Aux_State_val := ck_state_v( Vision_struct.States_in);
//read register from robot and chek is can read 2 or more correct values 
IF Aux_State_val = VCts.SeparatorRot_L_I THEN
	 I_STATE:= VCts.SeparatorRot_L_I;
//verifies that the vision system has completed its task
ELSIF Aux_State_val = VCts.SeparatorRot_L_F THEN
	//read the values processed by the vision system and send to robot
	sep_rot_left_data := ck_real_value(Vision_struct.Head_left_value);
	//check if all values are correct
	//IF sep_rot_left_data.Flag THEN
		//write variables from PLC to CS.UR5 Robot
		//IF wr_real_value(VCts.HEAD_LEFT_VALUE,sep_rot_left_data.Value) THEN
		    wr_real_value(VCts.HEAD_LEFT_VALUE,sep_rot_left_data.Value);
			I_STATE := VCts.SeparatorRot_L_F;
		//END_IF
	//END_IF
	
END_IF


//read internal variable and write over output variable
Act_In_State := I_STATE;
END_ACTION

ACTION CkHeadRot_L_entry:
//start the vision system
wr_state_v(Vcts.SeparatorRot_L);

//write the retain state variable 
Act_Gl_State:=VCts.SeparatorRot_L;
END_ACTION

ACTION CkHeadRot_L_exit:
//write reset state variables to visiom system.
wr_state_v(RCts.RESET_STATE);
//reset Global state variable
G_STATE := -1;
I_STATE :=-1;

//reset flags vision system to PLC
Vision_struct.States_in.Val1 := -1;
Vision_struct.States_in.Val2 := -1;
Vision_struct.States_in.Val3 := -1;
END_ACTION

ACTION CkHole_active:

Aux_State_val := ck_state_v( Vision_struct.States_in);
//read register from robot and chek is can read 2 or more correct values 
IF Aux_State_val = VCts.SeparatorHole_I THEN
	 I_STATE:= VCts.SeparatorHole_I;
//verifies that the vision system has completed its task
ELSIF Aux_State_val = VCts.SeparatorHole_F THEN
	//read the values processed by the vision system and send to robot
	cx_vision_data := ck_real_value(Vision_struct.Cx_value_hole);
	cy_vision_data := ck_real_value(Vision_struct.Cy_value_hole);
	
	//check if all values are correct
//	IF cx_vision_data.Flag AND cy_vision_data.Flag THEN
//		//write variables from PLC to CS.UR5 Robot
//		IF wr_real_value(VCts.CX_VALUE,cx_vision_data.Value) THEN
//			IF wr_real_value(VCts.CY_VALUE,cy_vision_data.Value) THEN				
//						I_STATE := VCts.SeparatorHole_F;
//			END_IF
		
//		END_IF
//	END_IF
	wr_real_value(VCts.CX_VALUE,cx_vision_data.Value);
	wr_real_value(VCts.CY_VALUE,cy_vision_data.Value);
	I_STATE := VCts.SeparatorHole_F;
	
END_IF




//read internal variable and write over output variable
Act_In_State := I_STATE;
END_ACTION

ACTION CkHole_entry:
//start the vision system
wr_state_v(Vcts.SeparatorHole);

//write the retain state variable 
Act_Gl_State:=VCts.SeparatorHole;
END_ACTION

ACTION CkHole_exit:
//write reset state variables to visiom system.
wr_state_v(RCts.RESET_STATE);
//reset Global state variable
G_STATE := -1;
I_STATE :=-1;


//reset flags vision system to PLC
Vision_struct.States_in.Val1 := -1;
Vision_struct.States_in.Val2 := -1;
Vision_struct.States_in.Val3 := -1;
END_ACTION

ACTION CkNut_active:

Aux_State_val := ck_state_v( Vision_struct.States_in);
//read register from robot and chek is can read 2 or more correct values 
IF Aux_State_val = VCts.SeparatorNut_I THEN
	 I_STATE:= VCts.SeparatorNut_I;
//verifies that the vision system has completed its task
ELSIF Aux_State_val = VCts.SeparatorNut_F  THEN
	//read the values processed by the vision system and send to robot
	cx_vision_data := ck_real_value(Vision_struct.Cx_value_nut);
	cy_vision_data := ck_real_value(Vision_struct.Cy_value_nut);
	nut_turn_data := ck_real_value(Vision_struct.Nut_turn_value);
	//check if all values are correct
	//IF cx_vision_data.Flag AND cy_vision_data.Flag AND nut_turn_data.Flag THEN
		//write variables from PLC to CS.UR5 Robot
		//I_STATE := VCts.SeparatorNut_F;
		wr_real_value(VCts.CX_VALUE,cx_vision_data.Value);
		wr_real_value(VCts.CY_VALUE,cy_vision_data.Value);
		wr_real_value(VCts.NUT_VALUE,nut_turn_data.Value);
		I_STATE := VCts.SeparatorNut_F;
		
		//IF wr_real_value(VCts.CX_VALUE,cx_vision_data.Value) THEN
		//	IF wr_real_value(VCts.CY_VALUE,cy_vision_data.Value) THEN
			//	IF wr_real_value(VCts.NUT_VALUE,nut_turn_data.Value) THEN
			//			I_STATE := VCts.SeparatorNut_F;
			//	END_IF
			//END_IF
		
		//END_IF
		
	//END_IF
	
END_IF



//read internal variable and write over output variable
Act_In_State := I_STATE;
END_ACTION

ACTION CkNut_entry:
//start the vision system
wr_state_v(Vcts.SeparatorNut);

//write the retain state variable 
Act_Gl_State:=VCts.SeparatorNut;
END_ACTION

ACTION CkNut_exit:

//write reset state variables to visiom system.
wr_state_v(RCts.RESET_STATE);
//reset Global state variable
G_STATE := -1;
//rest internat state variable
I_STATE :=-1;

//reset flags vision system to PLC
Vision_struct.States_in.Val1 := -1;
Vision_struct.States_in.Val2 := -1;
Vision_struct.States_in.Val3 := -1;
END_ACTION

ACTION CkPosSep_active:

Aux_State_val := ck_state_v( Vision_struct.States_in);
//read register from robot and chek is can read 2 or more correct values 
IF Aux_State_val = VCts.SeparatorPos_I THEN
	 I_STATE:= VCts.SeparatorPos_I;
	
//verifies that the vision system has completed its task
ELSIF  Aux_State_val = VCts.SeparatorPos_F THEN
	//I_STATE := VCts.SeparatorPos_F;
	//read the values processed by the vision system and send to robot
	sep_pos_data := ck_real_value(Vision_struct.Pos_sep);
	//check if all values are correct
	//IF sep_pos_data.Flag THEN
		//write variables from PLC to CS.UR5 Robot
		//IF wr_real_value(VCts.SEP_POS_VALUE,sep_pos_data.Value) THEN
		wr_real_value(VCts.SEP_POS_VALUE,sep_pos_data.Value);
		I_STATE := VCts.SeparatorPos_F;

		//END_IF
	//END_IF
	
END_IF

//read internal variable and write over output variable
Act_In_State := I_STATE;
END_ACTION

ACTION CkPosSep_entry:

//start the vision system
wr_state_v(Vcts.SeparatorPos);

//write the retain state variable 
Act_Gl_State:=VCts.SeparatorPos;
END_ACTION

ACTION CkPosSep_exit:

//write reset state variables to visiom system.
wr_state_v(RCts.RESET_STATE);
//reset Global state variable
G_STATE := -1;
//rest internat state variable
I_STATE :=-1;

//reset flags vision system to PLC
Vision_struct.States_in.Val1 := -1;
Vision_struct.States_in.Val2 := -1;
Vision_struct.States_in.Val3 := -1;
END_ACTION

ACTION Wrt_FState_entry:
//write output variable to indicate that the robot execute the state 
State_complete := TRUE;
END_ACTION

ACTION Wrt_FState_exit:
//write output variable to indicate that the robot execute the state 
State_complete := FALSE;
//init_:=FALSE;

G_STATE := -1;
//rest internat state variable
I_STATE :=-1;
END_ACTION

END_PROGRAM

// ---- POUs/POUs/VISION/Vision_functions/ck_state_v.TcPOU
FUNCTION ck_state_v : INT
VAR_INPUT
	
	data_vision : Vision_int_state;
    
END_VAR
VAR
	ck0 : INT;
	ck1 : INT;
	ck2 : INT;
END_VAR


ck0 := data_vision.Val1;
ck1 := data_vision.Val2;
ck2 := data_vision.Val3;


//IF (ck0=state AND ck1=state AND ck2=state) OR (ck1=state AND ck2=state) OR (ck0=state AND ck2=state) OR (ck0=state AND ck1=state ) THEN
IF ck0 = ck1 THEN
ck_state_v := ck0;	
ELSIF  ck1 = ck2 THEN 
ck_state_v := ck1;	
ELSIF  ck2 = ck0 THEN
ck_state_v := ck2;	
ELSE 
ck_state_v := -1;	
END_IF

END_FUNCTION

// ---- POUs/POUs/VISION/Vision_functions/ck_real_value.TcPOU
FUNCTION ck_real_value :ck_real_flag_data
//return ck_real_flag_data struct
VAR_INPUT
	//imput Vision_data struct 
	data: Vision_data;
END_VAR
VAR
END_VAR


//check if two of tree values are the same, to avoid bad variables intercahnages between vision system and plc
//return flag ck_real_flag_data[0] to indicate is correct, and one real value ck_real_value[1] 
IF data.Val2=data.Val3 THEN
	ck_real_value.Flag:=TRUE;
	ck_real_value.Value:=data.Val2;
ELSIF data.Val1=data.Val3 THEN
	ck_real_value.Flag:=TRUE;
	ck_real_value.Value:=data.Val3;
ELSIF data.Val1=data.Val2 THEN
	ck_real_value.Flag:=TRUE;
	ck_real_value.Value:=data.Val2;
ELSIF (data.Val1=data.Val2 AND data.Val1=data.Val3 AND data.Val2=data.Val3) THEN	
	ck_real_value.Flag:=TRUE;
	ck_real_value.Value:=data.Val1;
ELSE	
	ck_real_value.Flag:=FALSE;
	ck_real_value.Value:=-1;
END_IF

END_FUNCTION

// ---- POUs/POUs/VISION/Vision_functions/wr_state_v.TcPOU
FUNCTION wr_state_v : BOOL
VAR_INPUT
	state : INT;
END_VAR
VAR
END_VAR

wr_state_v := FALSE;
//WRITE FLAGS STATE-MACHINE #################(PLC->VISION SYSTEM)
Vision_struct.States_out.Val1:=state;
Vision_struct.States_out.Val2:=state;
Vision_struct.States_out.Val3:=state;
wr_state_v := TRUE;

END_FUNCTION

// ---- POUs/POUs/Qrob/Qrob_State_Machine/QRob_StateMachine.TcPOU
PROGRAM QRob_StateMachine
VAR_INPUT
init_: BOOL:= True;
//global aux state
G_STATE : INT := -1;
//comaper position to stop
Position : LREAL:= 0;
Velocity : REAL:=170;
Torque : INT := 0;
Torque_ramp : INT := 100;
Control :E_DRIVEOPERATIONMODE;
Reset_State : BOOL:= FALSE;
//Max_profile_velocity AT%Q*:UDINT := 314572;
//Modes_operation AT%Q*:USINT:= 8;
//actual_torque AT%I*:INT ;

//Qrob_set torque 
torquevalut AT%Q*:INT;


END_VAR
VAR_OUTPUT
	State_complete : BOOL := FALSE;
	Act_Gl_State : INT := -1;
	Act_In_State : INT := -1;
	Act_Pos : LREAL := -1;
END_VAR
VAR
	
//Axis status
Axis_state :BOOL:=FALSE;
	//internal aux state
I_STATE : INT:=-1;
Aux_error :INT:=-1;
//blocks to activate axis of qrob
Reset : MC_Reset;
ResetOut: ST_McOutputs;

PowerAxis1 : MC_Power;
/// debug function block output data 
PowerAxis1Out: ST_McOutputs;



//blocks to move axis 
MoveAbsAxis1 :MC_MoveAbsolute;
MoveAbsoluteOut1: ST_McOutputs;

//block to set home position
Home : MC_Home;
HomeOut: ST_McOutputs;

//block to read and change the contyrol mode
WriteDriveOperationMode : MC_WriteDriveOperationMode;
WDO_ModeOut : ST_McOutputs;

ReadDriveOperationMode : MC_ReadDriveOperationMode;
RDO_ModeOut : ST_McOutputs;
ReadOperation_mode : E_DRIVEOPERATIONMODE;

//block to Control Mode
TorqueControl : MC_TorqueControl;
TorqueControlOut : ST_McOutputs;
Torque_done : BOOL;
Qrob_velocity AT%I*:DINT := -1;
Qrob_torque AT%I*:INT := -1;

//block stop motion
Stop : MC_Stop;
StopOut: ST_McOutputs;

//var to ck torque done
F_vel : BOOL ;
F_tor : BOOL;
F_tor_done : BOOL;


//var to offfset Home
offset_home :INT := 3;
offset_flag : INT := -1;

Sensor_Position_detection AT%I*: BOOL;


END_VAR

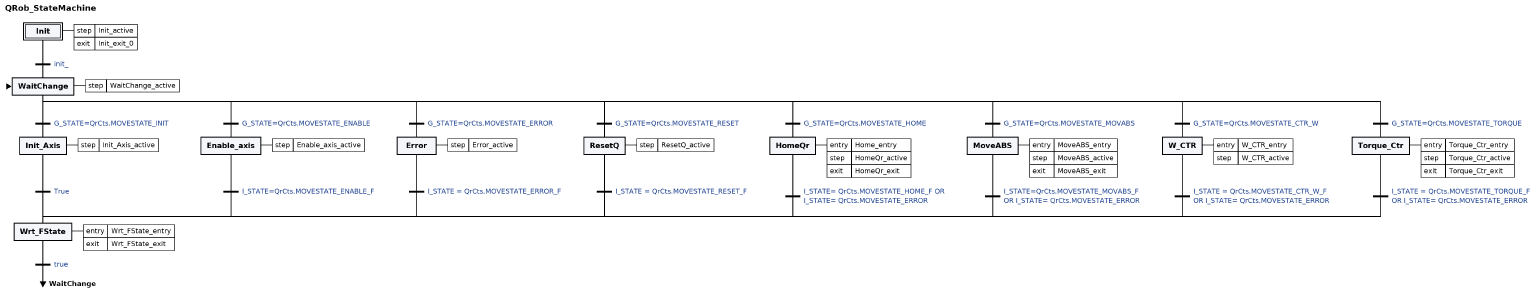
INITIAL_STEP Init:
    Init_active(N);  // step action
    Init_exit_0(P0);  // exit action
END_STEP
TRANSITION FROM Init TO WaitChange
    := init_;
END_TRANSITION
STEP WaitChange:
    WaitChange_active(N);  // step action
END_STEP
TRANSITION FROM WaitChange TO Init_Axis
    := G_STATE=QrCts.MOVESTATE_INIT;
END_TRANSITION
STEP Init_Axis:
    Init_Axis_active(N);  // step action
END_STEP
TRANSITION FROM Init_Axis TO Wrt_FState
    := True;
END_TRANSITION
TRANSITION FROM WaitChange TO Enable_axis
    := G_STATE=QrCts.MOVESTATE_ENABLE;
END_TRANSITION
STEP Enable_axis:
    Enable_axis_active(N);  // step action
END_STEP
TRANSITION FROM Enable_axis TO Wrt_FState
    := I_STATE=QrCts.MOVESTATE_ENABLE_F;
END_TRANSITION
TRANSITION FROM WaitChange TO Error
    := G_STATE=QrCts.MOVESTATE_ERROR;
END_TRANSITION
STEP Error:
    Error_active(N);  // step action
END_STEP
TRANSITION FROM Error TO Wrt_FState
    := I_STATE = QrCts.MOVESTATE_ERROR_F;
END_TRANSITION
TRANSITION FROM WaitChange TO ResetQ
    := G_STATE=QrCts.MOVESTATE_RESET;
END_TRANSITION
STEP ResetQ:
    ResetQ_active(N);  // step action
END_STEP
TRANSITION FROM ResetQ TO Wrt_FState
    := I_STATE = QrCts.MOVESTATE_RESET_F;
END_TRANSITION
TRANSITION FROM WaitChange TO HomeQr
    := G_STATE=QrCts.MOVESTATE_HOME;
END_TRANSITION
STEP HomeQr:
    Home_entry(P1);  // entry action
    HomeQr_active(N);  // step action
    HomeQr_exit(P0);  // exit action
END_STEP
TRANSITION FROM HomeQr TO Wrt_FState
    := I_STATE= QrCts.MOVESTATE_HOME_F OR I_STATE= QrCts.MOVESTATE_ERROR;
END_TRANSITION
TRANSITION FROM WaitChange TO MoveABS
    := G_STATE=QrCts.MOVESTATE_MOVABS;
END_TRANSITION
STEP MoveABS:
    MoveABS_entry(P1);  // entry action
    MoveABS_active(N);  // step action
    MoveABS_exit(P0);  // exit action
END_STEP
TRANSITION FROM MoveABS TO Wrt_FState
    := I_STATE=QrCts.MOVESTATE_MOVABS_F OR I_STATE= QrCts.MOVESTATE_ERROR;
END_TRANSITION
TRANSITION FROM WaitChange TO W_CTR
    := G_STATE=QrCts.MOVESTATE_CTR_W;
END_TRANSITION
STEP W_CTR:
    W_CTR_entry(P1);  // entry action
    W_CTR_active(N);  // step action
END_STEP
TRANSITION FROM W_CTR TO Wrt_FState
    := I_STATE = QrCts.MOVESTATE_CTR_W_F OR I_STATE= QrCts.MOVESTATE_ERROR;
END_TRANSITION
TRANSITION FROM WaitChange TO Torque_Ctr
    := G_STATE=QrCts.MOVESTATE_TORQUE;
END_TRANSITION
STEP Torque_Ctr:
    Torque_Ctr_entry(P1);  // entry action
    Torque_Ctr_active(N);  // step action
    Torque_Ctr_exit(P0);  // exit action
END_STEP
TRANSITION FROM Torque_Ctr TO Wrt_FState
    := I_STATE = QrCts.MOVESTATE_TORQUE_F OR I_STATE= QrCts.MOVESTATE_ERROR;
END_TRANSITION
STEP Wrt_FState:
    Wrt_FState_entry(P1);  // entry action
    Wrt_FState_exit(P0);  // exit action
END_STEP
TRANSITION FROM Wrt_FState TO WaitChange
    := true;
END_TRANSITION

ACTION AC_WriteControl:
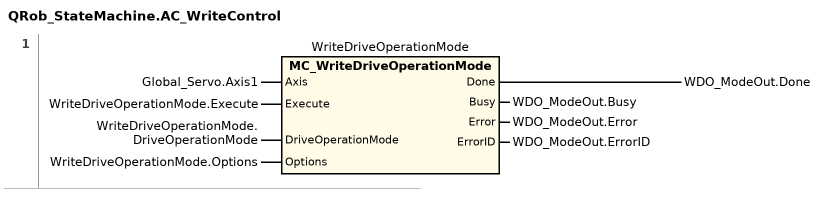
// NETWORK 1
WriteDriveOperationMode(
    Axis := Global_Servo.Axis1,
    Execute := WriteDriveOperationMode.Execute,
    DriveOperationMode := WriteDriveOperationMode.DriveOperationMode,
    Options := WriteDriveOperationMode.Options,
    Busy => WDO_ModeOut.Busy,
    Error => WDO_ModeOut.Error,
    ErrorID => WDO_ModeOut.ErrorID); // MC_WriteDriveOperationMode
WDO_ModeOut.Done := WriteDriveOperationMode.Done;
END_ACTION

ACTION Act_Home:
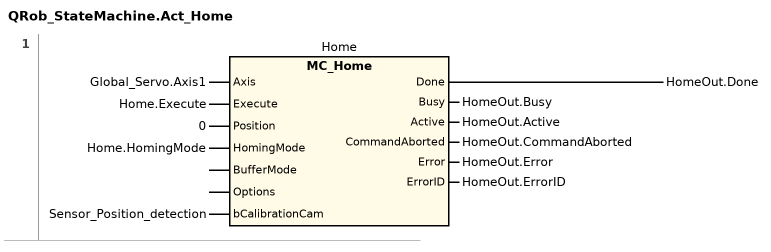
// NETWORK 1
Home(
    Axis := Global_Servo.Axis1,
    Execute := Home.Execute,
    Position := 0,
    HomingMode := Home.HomingMode,
    bCalibrationCam := Sensor_Position_detection,
    Busy => HomeOut.Busy,
    Active => HomeOut.Active,
    CommandAborted => HomeOut.CommandAborted,
    Error => HomeOut.Error,
    ErrorID => HomeOut.ErrorID); // MC_Home
HomeOut.Done := Home.Done;
END_ACTION

ACTION Act_MoveAbs:
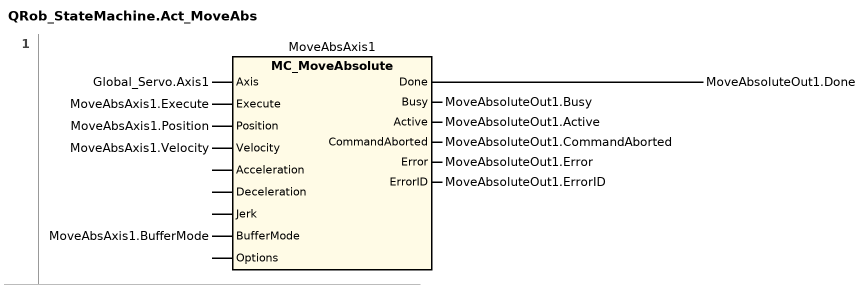
// NETWORK 1
MoveAbsAxis1(
    Axis := Global_Servo.Axis1,
    Execute := MoveAbsAxis1.Execute,
    Position := MoveAbsAxis1.Position,
    Velocity := MoveAbsAxis1.Velocity,
    BufferMode := MoveAbsAxis1.BufferMode,
    Busy => MoveAbsoluteOut1.Busy,
    Active => MoveAbsoluteOut1.Active,
    CommandAborted => MoveAbsoluteOut1.CommandAborted,
    Error => MoveAbsoluteOut1.Error,
    ErrorID => MoveAbsoluteOut1.ErrorID); // MC_MoveAbsolute
MoveAbsoluteOut1.Done := MoveAbsAxis1.Done;
END_ACTION

ACTION Act_Power:
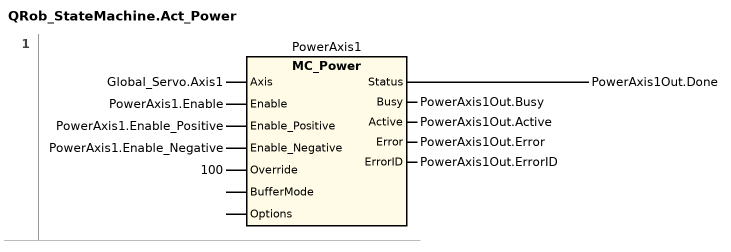
// NETWORK 1
PowerAxis1(
    Axis := Global_Servo.Axis1,
    Enable := PowerAxis1.Enable,
    Enable_Positive := PowerAxis1.Enable_Positive,
    Enable_Negative := PowerAxis1.Enable_Negative,
    Override := 100,
    Busy => PowerAxis1Out.Busy,
    Active => PowerAxis1Out.Active,
    Error => PowerAxis1Out.Error,
    ErrorID => PowerAxis1Out.ErrorID); // MC_Power
PowerAxis1Out.Done := PowerAxis1.Status;
END_ACTION

ACTION Act_ReadControl:
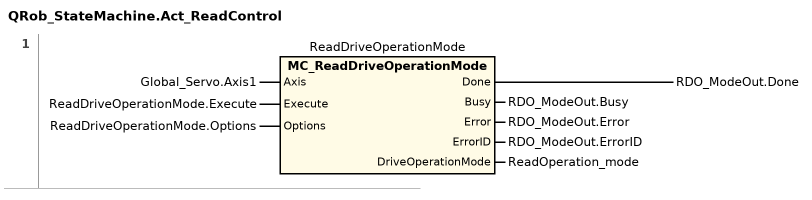
// NETWORK 1
ReadDriveOperationMode(
    Axis := Global_Servo.Axis1,
    Execute := ReadDriveOperationMode.Execute,
    Options := ReadDriveOperationMode.Options,
    Busy => RDO_ModeOut.Busy,
    Error => RDO_ModeOut.Error,
    ErrorID => RDO_ModeOut.ErrorID,
    DriveOperationMode => ReadOperation_mode); // MC_ReadDriveOperationMode
RDO_ModeOut.Done := ReadDriveOperationMode.Done;
END_ACTION

ACTION Act_Reset:
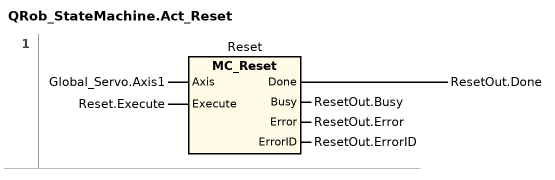
// NETWORK 1
Reset(
    Axis := Global_Servo.Axis1,
    Execute := Reset.Execute,
    Busy => ResetOut.Busy,
    Error => ResetOut.Error,
    ErrorID => ResetOut.ErrorID); // MC_Reset
ResetOut.Done := Reset.Done;
END_ACTION

ACTION Act_Stop:
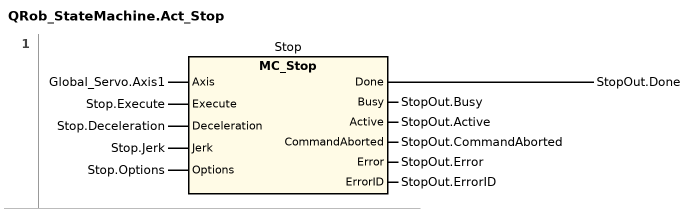
// NETWORK 1
Stop(
    Axis := Global_Servo.Axis1,
    Execute := Stop.Execute,
    Deceleration := Stop.Deceleration,
    Jerk := Stop.Jerk,
    Options := Stop.Options,
    Busy => StopOut.Busy,
    Active => StopOut.Active,
    CommandAborted => StopOut.CommandAborted,
    Error => StopOut.Error,
    ErrorID => StopOut.ErrorID); // MC_Stop
StopOut.Done := Stop.Done;
END_ACTION

ACTION Act_Torque:
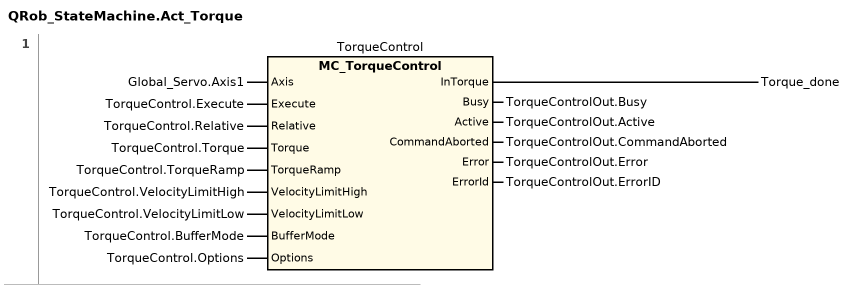
// NETWORK 1
TorqueControl(
    Axis := Global_Servo.Axis1,
    Execute := TorqueControl.Execute,
    Relative := TorqueControl.Relative,
    Torque := TorqueControl.Torque,
    TorqueRamp := TorqueControl.TorqueRamp,
    VelocityLimitHigh := TorqueControl.VelocityLimitHigh,
    VelocityLimitLow := TorqueControl.VelocityLimitLow,
    BufferMode := TorqueControl.BufferMode,
    Options := TorqueControl.Options,
    Busy => TorqueControlOut.Busy,
    Active => TorqueControlOut.Active,
    CommandAborted => TorqueControlOut.CommandAborted,
    Error => TorqueControlOut.Error,
    ErrorId => TorqueControlOut.ErrorID); // MC_TorqueControl
Torque_done := TorqueControl.InTorque;
END_ACTION

ACTION Enable_axis_active:
//power on axis
PowerAxis1.Enable := TRUE;
PowerAxis1.Enable_Positive := TRUE;
PowerAxis1.Enable_Negative := TRUE;


IF PowerAxis1.Status THEN
//check the state where the error is produced	
	CASE Aux_error OF 
		QrCts.MOVESTATE_MOVABS:
			G_STATE := QrCts.MOVESTATE_MOVABS;
		QrCts.MOVESTATE_HOME:
			G_STATE := QrCts.MOVESTATE_HOME;
		QrCts.MOVESTATE_CTR_W:
			G_STATE := QrCts.MOVESTATE_CTR_W;
		QrCts.MOVESTATE_TORQUE:	
			G_STATE := QrCts.MOVESTATE_TORQUE;
		QrCts.MOVESTATE_RELIEF:
			G_STATE := QrCts.MOVESTATE_RELIEF;
	ELSE
		G_STATE := -1;
	END_CASE
	I_STATE := QrCts.MOVESTATE_ENABLE_F;
ELSIF PowerAxis1.Error THEN
	G_STATE := QrCts.MOVESTATE_ERROR;
	I_STATE := QrCts.MOVESTATE_ENABLE_F;
END_IF

(* call the power function block *)
Act_Power();
Act_Reset();
Act_MoveAbs();
END_ACTION

ACTION Enable_axis_entry:
//power on axis
PowerAxis1.Enable := TRUE;
PowerAxis1.Enable_Positive := TRUE;
PowerAxis1.Enable_Negative := TRUE;
END_ACTION

ACTION Error_active:
IF Global_Servo.Axis1.NcToPlc.ErrorCode <>0 THEN
	G_STATE := QrCts.MOVESTATE_RESET;	(* axis error requires reset *)
	I_STATE := QrCts.MOVESTATE_ERROR_F;
ELSE
G_STATE := QrCts.MOVESTATE_INIT;
I_STATE := QrCts.MOVESTATE_ERROR_F;		(* function block errors don't need a reset *)
END_IF


(* call the power function block *)
Act_Power();
Act_Reset();
Act_MoveAbs();
END_ACTION

ACTION Home_entry:

//start fuction block 
Home.Execute := TRUE;

IF offset_flag = 1 THEN 
	Home.HomingMode := MC_Direct;
	offset_flag := offset_flag +1 ;
ELSE  	
	Home.HomingMode := MC_DefaultHoming;
END_IF


//write the retain state variable 
Act_Gl_State:=QrCts.MOVESTATE_HOME;
//read internal variable and write over output variable
I_STATE := QrCts.MOVESTATE_HOME_I;
Act_In_State := I_STATE;
END_ACTION

ACTION HomeQr_active:



//Home.bCalibrationCam := Sensor_Position_detection; 

IF Home.CommandAborted OR Home.Error THEN
	G_STATE := QrCts.MOVESTATE_ERROR;
	I_STATE := QrCts.MOVESTATE_ERROR;
	Aux_error := QrCts.MOVESTATE_HOME;
	Act_In_State := I_STATE;
ELSIF Home.Done THEN
	I_STATE := QrCts.MOVESTATE_HOME_F;
	//read internal variable and write over output variable
	Act_In_State := I_STATE;
	G_STATE := QrCts.MOVESTATE_MOVABS;
	position := offset_home;
	Home.Execute := FALSE; 
  IF offset_flag >= 2 THEN
	  G_STATE := -1;
	  offset_flag := -1;
  ELSE
	  G_STATE := QrCts.MOVESTATE_MOVABS;
	  offset_flag := offset_flag + 1;
  END_IF
	
END_IF





(* call the power function block *)
Act_Power();
Act_Reset();
Act_Home();
Act_MoveAbs();
END_ACTION

ACTION HomeQr_exit:
I_STATE :=-1;
END_ACTION

ACTION Init_active:

END_ACTION

ACTION Init_Axis_active:


//star variables
MoveAbsAxis1.Execute := FALSE;
Reset.Execute := FALSE;
Home.Execute := FALSE;
//write the global staus
G_State := QrCts.MOVESTATE_ENABLE;




(* call the power function block *)
Act_Power();
Act_Reset();
Act_MoveAbs();
Act_Home();
END_ACTION

ACTION Init_Axis_entry:

END_ACTION

ACTION Init_Axis_exit:

END_ACTION

ACTION Init_exit:
// NETWORK 1
END_ACTION

ACTION Init_exit_0:
G_STATE:=QrCts.MOVESTATE_INIT;


//check is there are some error
IF Global_Servo.Axis1.NcToPlc.ErrorCode <>0 THEN
	G_STATE := QrCts.MOVESTATE_RESET;	(* axis error requires reset *)
	
//ELSE
//	G_STATE := QrCts.MOVESTATE_INIT;
//	I_STATE := QrCts.MOVESTATE_ERROR_F;		(* function block errors don't need a reset *)
END_IF
END_ACTION

ACTION MoveABS_active:


IF MoveAbsAxis1.CommandAborted OR MoveAbsAxis1.Error THEN
	G_STATE := QrCts.MOVESTATE_ERROR;
	I_STATE := QrCts.MOVESTATE_ERROR;
	Aux_error := QrCts.MOVESTATE_MOVABS;
	Position := Position - Act_Pos;
	//read internal variable and write over output variable
	Act_In_State := I_STATE;
ELSIF MoveAbsAxis1.Done THEN
	I_STATE := QrCts.MOVESTATE_MOVABS_F;
	//read internal variable and write over output variable
	Act_In_State := I_STATE;
	G_STATE := -1;
	MoveAbsAxis1.Execute := FALSE;
ELSIF Reset_state THEN
	I_STATE := QrCts.MOVESTATE_MOVABS_F;;
	Act_In_State := I_STATE;
	G_STATE := -1;
	
	Stop.Execute := TRUE;
    MoveAbsAxis1.Execute := FALSE;	
	Reset_state := FALSE;
END_IF


//read actual postion
Act_Pos := Global_Servo.Axis1.NcToPlc.ActPos;

(* call the power function block *)
Act_Power();
Act_Reset();
Act_MoveAbs();
Act_Stop();
END_ACTION

ACTION MoveABS_entry:

MoveAbsAxis1.Position := Position;
MoveAbsAxis1.Velocity := Velocity;
//MoveAbsAxis1.BufferMode := MC_Buffered;
MoveAbsAxis1.Execute := TRUE;



//write the retain state variable 
Act_Gl_State:=QrCts.MOVESTATE_MOVABS;
//read internal variable and write over output variable
I_STATE := QrCts.MOVESTATE_MOVABS_I;
Act_In_State := I_STATE;

(* call the power function block *)
Act_Power();
Act_Reset();
Act_MoveAbs();
Act_Stop();
END_ACTION

ACTION MoveABS_exit:

//condition to execute home position
IF offset_flag = 0 THEN 
	G_STATE := QrCts.MOVESTATE_HOME;
    offset_flag := offset_flag +1 ;
END_IF


I_STATE :=-1;


Stop.Execute := FALSE;
Reset_state := FALSE;


(* call the power function block *)
Act_Power();
Act_Reset();
Act_MoveAbs();
Act_Stop();
END_ACTION

ACTION ResetQ_active:
WriteDriveOperationMode.Execute := FALSE;
Home.Execute := FALSE;
ReadDriveOperationMode.Execute := FALSE;
Stop.Execute := FALSE;
MoveAbsAxis1.Execute := FALSE;
TorqueControl.Execute := FALSE;
Stop.Execute := FALSE; 

Reset.Execute := TRUE;


IF Reset.Done THEN
	G_STATE := QrCts.MOVESTATE_INIT;
	I_STATE := QrCts.MOVESTATE_RESET_F;
ELSIF Reset.Error THEN
	G_STATE := QrCts.MOVESTATE_INIT; (* can't do anything here *)
	//I_STATE := QrCts.MOVESTATE_RESET_F;
END_IF


(* call the power function block *)
Act_Power();
Act_Reset();
Act_MoveAbs();
Act_Stop();
END_ACTION

ACTION Sleep_exit:
TorqueControl.Execute := False;
END_ACTION

ACTION Torque_Ctr_active:
IF TorqueControlOut.CommandAborted OR TorqueControlOut.Error THEN
	G_STATE := QrCts.MOVESTATE_ERROR;
	I_STATE := QrCts.MOVESTATE_ERROR;
	Aux_error := QrCts.MOVESTATE_TORQUE;
	//read internal variable and write over output variable
	Act_In_State := I_STATE;
ELSIF Torque_done THEN
	F_tor_done := TRUE;
END_IF



IF Qrob_torque = Torque THEN 
	F_tor := TRUE;
		IF Qrob_velocity <=0  THEN 
			F_vel := TRUE;
	END_IF
END_IF


IF F_vel AND F_tor AND F_tor_done THEN

	I_STATE := QrCts.MOVESTATE_TORQUE_F;
	//read internal variable and write over output variable
	Act_In_State := I_STATE;
	G_STATE := -1;
	TorqueControl.Execute := FALSE;
	Torque_done := FALSE;
	
	F_vel  := FALSE;
	F_tor  := FALSE;
	F_tor_done  := FALSE;
	//I_STATE :=-1;	

END_IF

(* call the power function block *)
Act_Power();
Act_Reset();
Act_MoveAbs();
Act_Torque();
END_ACTION

ACTION Torque_Ctr_entry:
// write the variables TorqueControl block function
TorqueControl.Relative := FALSE;
TorqueControl.Torque := Torque;
torquevalut := Torque;
TorqueControl.TorqueRamp := 100;
TorqueControl.VelocityLimitHigh := 100;
TorqueControl.VelocityLimitLow := 1;
TorqueControl.Execute := True;


//write the retain state variable 
Act_Gl_State:=QrCts.MOVESTATE_TORQUE;
//read internal variable and write over output variable
I_STATE := QrCts.MOVESTATE_TORQUE_I;
Act_In_State := I_STATE;
END_ACTION

ACTION Torque_Ctr_exit:
	TorqueControl.Execute := FALSE;
	Torque_done := FALSE;
	//I_STATE :=-1;
	//G_STATE := -1;
	
	I_STATE :=-1;
END_ACTION

ACTION Torque_Relie_active:
//ggggggggggggggg


IF TorqueControlOut.CommandAborted OR TorqueControlOut.Error THEN
	G_STATE := QrCts.MOVESTATE_ERROR;
	I_STATE := QrCts.MOVESTATE_ERROR;
	Aux_error := QrCts.MOVESTATE_RELIEF;
	//read internal variable and write over output variable
	Act_In_State := I_STATE;
ELSIF Torque_done THEN
	F_tor_done := TRUE;
END_IF

//F_tor_done := TRUE;

IF Qrob_torque = 0 THEN 
	F_tor := TRUE;
		IF (-5 <= Qrob_velocity) AND  (Qrob_velocity<= 5) THEN 
			F_vel := TRUE;
	END_IF
END_IF


IF F_vel AND F_tor AND F_tor_done THEN

	I_STATE := QrCts.MOVESTATE_RELIEF_F;
	//read internal variable and write over output variable
	Act_In_State := I_STATE;
	G_STATE := -1;
	TorqueControl.Execute := TRUE;
	Torque_done := FALSE;
	
	F_vel  := FALSE;
	F_tor  := FALSE;
	F_tor_done  := FALSE;
	//I_STATE :=-1;	

END_IF

(* call the power function block *)
Act_Power();
Act_Reset();
Act_MoveAbs();
Act_Torque();
END_ACTION

ACTION Torque_Relie_entry:
// write the variables TorqueControl block function
TorqueControl.Relative := FALSE;
TorqueControl.Torque := 0;
TorqueControl.TorqueRamp := 0;
TorqueControl.VelocityLimitHigh := 100;
TorqueControl.VelocityLimitLow := 0;
//torquevalut := 0;
TorqueControl.Execute := True;


//write the retain state variable 
Act_Gl_State:=QrCts.MOVESTATE_RELIEF;
//read internal variable and write over output variable
I_STATE := QrCts.MOVESTATE_RELIEF_I;
Act_In_State := I_STATE;
END_ACTION

ACTION Torque_Relie_exit:
	TorqueControl.Execute := FALSE;
	Torque_done := FALSE;
	
	I_STATE :=-1;
END_ACTION

ACTION W_CTR_active:
IF WriteDriveOperationMode.Error THEN
	G_STATE := QrCts.MOVESTATE_ERROR;
	I_STATE := QrCts.MOVESTATE_ERROR;
	Aux_error := QrCts.MOVESTATE_CTR_W;
	//read internal variable and write over output variable
	Act_In_State := I_STATE;
ELSIF WriteDriveOperationMode.Done THEN
	//Read if the control mode have been change
	ReadDriveOperationMode.Execute := TRUE;
	IF ReadDriveOperationMode.Error THEN
		G_STATE := QrCts.MOVESTATE_ERROR;
		I_STATE := QrCts.MOVESTATE_ERROR;
		Aux_error := QrCts.MOVESTATE_CTR_W;
		//read internal variable and write over output variable
		Act_In_State := I_STATE;
	 	ReadDriveOperationMode.Execute := FALSE; 
	
	ELSIF ReadDriveOperationMode.Done THEN
		
		IF ReadOperation_mode = Control THEN

			I_STATE := QrCts.MOVESTATE_CTR_W_F;
			//read internal variable and write over output variable
			Act_In_State := I_STATE;
			//G_STATE := -1;
			WriteDriveOperationMode.Execute := FALSE;
			ReadDriveOperationMode.Execute := FALSE; 
			G_STATE := QrCts.MOVESTATE_RESET;
			//I_STATE :=-1;
		END_IF
		ReadDriveOperationMode.Execute := FALSE; 
	END_IF
END_IF


(* call the  function block *)
Act_Power();
Act_Reset();
AC_WriteControl();
Act_ReadControl();
END_ACTION

ACTION W_CTR_entry:
WriteDriveOperationMode.DriveOperationMode := Control;
WriteDriveOperationMode.Execute := TRUE;

//write the retain state variable 
Act_Gl_State:=QrCts.MOVESTATE_CTR_W;
//read internal variable and write over output variable
I_STATE := QrCts.MOVESTATE_CTR_W_I;
Act_In_State := I_STATE;
END_ACTION

ACTION WaitChange_active:

END_ACTION

ACTION Wrt_FState_entry:
//write output variable to indicate that the robot execute the state 
State_complete := TRUE;
END_ACTION

ACTION Wrt_FState_exit:
//write output variable to indicate that the robot execute the state 
State_complete := FALSE;
Reset_State := FALSE;
END_ACTION

END_PROGRAM

// ---- POUs/POUs/ROBOTS/Robot_functions/read_bool_flag_move.TcPOU
FUNCTION read_bool_flag_move : BOOL
VAR_INPUT

	state : BOOL;
END_VAR
VAR
	ck0 : BOOL;
	ck1 : BOOL;
	ck2 : BOOL;
END_VAR

//Read bit register from Robot to PLC
ck0 := Robot_UR5.UR_outputs.B3;
ck1 := Robot_UR5.UR_outputs.B4;
ck2 := Robot_UR5.UR_outputs.B5;

IF (ck0=state AND ck1=state AND ck2=state) OR (ck0<>state AND ck1=state AND ck2=state) OR (ck0=state AND ck1<>state AND ck2=state) OR (ck0=state AND ck1=state AND ck2<>state) THEN
read_bool_flag_move := TRUE;
ELSE 
read_bool_flag_move := FALSE;	
END_IF

END_FUNCTION

// ---- POUs/POUs/ROBOTS/Robot_functions/read_bool_flag.TcPOU
FUNCTION read_bool_flag : BOOL
VAR_INPUT

	state : BOOL;
END_VAR
VAR
	ck0 : BOOL;
	ck1 : BOOL;
	ck2 : BOOL;
END_VAR

//Read bit register from Robot to PLC
ck0 := Robot_UR5.UR_outputs.B0;
ck1 := Robot_UR5.UR_outputs.B1;
ck2 := Robot_UR5.UR_outputs.B2;

IF (ck0=state AND ck1=state AND ck2=state) OR (ck0<>state AND ck1=state AND ck2=state) OR (ck0=state AND ck1<>state AND ck2=state) OR (ck0=state AND ck1=state AND ck2<>state) THEN
read_bool_flag := TRUE;
ELSE 
read_bool_flag := FALSE;	
END_IF

END_FUNCTION

// ---- POUs/POUs/Qrob/QRob_functions/Get_QRob_Pos.TcPOU
PROGRAM Get_QRob_Pos
VAR
	
MC_ReadActualPosition : MC_ReadActualPosition;
actual_position : REAL;

Driver_temperature_C AT%I*:UINT:= 0;


    FB_CoERead_ByDriveRef : FB_CoERead_ByDriveRef;
    stDriveRef        :  ST_DriveRef := (sNetId:= '172.18.236.0.6.1', nDriveNo := 1, nDriveType := 16, nSlaveAddr := 1001); 

    Index             : WORD := 16#22A2;
    SubIndex          : BYTE := 0; 
    Execute           : BOOL := TRUE;
    Timeout           : TIME := T#5S;
    CompleteAccess    : BOOL := TRUE;
    vendorId          : UINT ;
    Error             : BOOL;
    AdsErrId          : UDINT;
    CANopenErrId      : UDINT;
	
	FB_EcCoESdoRead : FB_EcCoESdoRead;
	dir :  T_AmsNetId := '172.18.236.0.6.1';
	
	pSample : POINTER TO UINT;
	driver_temperature : UINT;
	
	Cooler_fan AT%Q*:BOOL:= FALSE;
	Temperature_Ctr : Temperature_Ctr;

END_VAR

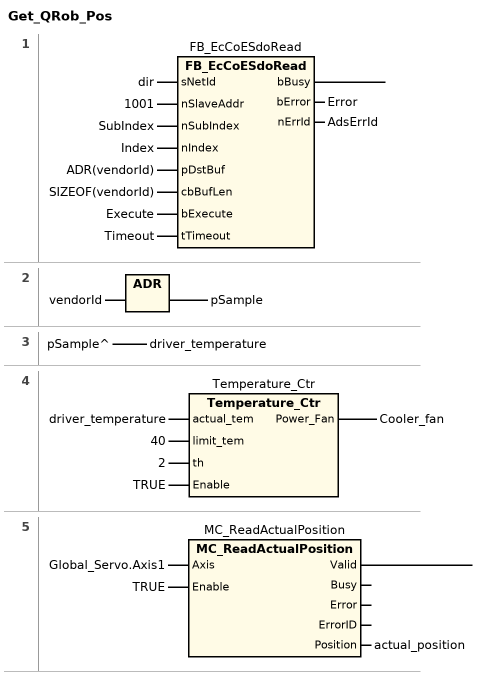
// NETWORK 1
FB_EcCoESdoRead(
    sNetId := dir,
    nSlaveAddr := 1001,
    nSubIndex := SubIndex,
    nIndex := Index,
    pDstBuf := ADR(vendorId),
    cbBufLen := SIZEOF(vendorId),
    bExecute := Execute,
    tTimeout := Timeout,
    bError => Error,
    nErrId => AdsErrId);

// NETWORK 2
pSample := ADR(vendorId);

// NETWORK 3
driver_temperature := pSample^;

// NETWORK 4
Temperature_Ctr(actual_tem := driver_temperature, limit_tem := 40, th := 2, Enable := TRUE);
Cooler_fan := Temperature_Ctr.Power_Fan;

// NETWORK 5
MC_ReadActualPosition(Axis := Global_Servo.Axis1, Enable := TRUE, Position => actual_position);

END_PROGRAM

// ---- POUs/POUs/Qrob/QRob_functions/Temperature_Ctr.TcPOU
FUNCTION_BLOCK Temperature_Ctr
VAR_INPUT
	actual_tem : REAL;
	limit_tem : REAL;
	th : REAL;
	Enable : BOOL;	
	
	//relief_turn : BOOL := FALSE;	
   
	
END_VAR
VAR_OUTPUT
	Power_Fan :BOOL;
END_VAR
VAR
	A : REAL;
	B : REAL;
	
END_VAR


IF Enable = TRUE THEN 
	A := limit_tem-th;
	B := limit_tem +th;
	
	IF (actual_tem <= A)  THEN 
		Power_Fan := FALSE;
	ELSIF (actual_tem >= B) THEN
		Power_Fan := TRUE;
	END_IF
END_IF

END_FUNCTION_BLOCK

// ---- POUs/POUs/Fuzzy/Subsystem.TcPOU
FUNCTION_BLOCK Subsystem
VAR_INPUT
	in: LREAL;
	state : BOOL;
END_VAR
VAR_OUTPUT
	out: LREAL;
	set_move  : BOOL := TRUE;
	
END_VAR
VAR
	
  	state_aux : BOOL := FALSE;	
	before_out : INT;
	aux : INT := 0;
out_int : INT;


	ruleID: DINT;
	y1: LREAL;
	y2: LREAL;
	outputMFCache: ARRAY[0..302] OF LREAL;
	sampleID: DINT;
	rtb_antecedentOutputs: ARRAY[0..2] OF LREAL;
	rtb_aggregatedOutputs: ARRAY[0..100] OF LREAL;
	tmp: ARRAY[0..100] OF LREAL;
	tmp_0: ARRAY[0..100] OF LREAL;
	tmp_1: ARRAY[0..100] OF LREAL;
	inputMFCache_idx_1: LREAL;
	inputMFCache_idx_2: LREAL;
	i0_trimf_l: trimf_l;
	OutputSamplePoints_Value: ARRAY[0..100] OF LREAL := [0.0, 1.5, 3.0, 4.5, 6.0, 7.5, 9.0, 10.5, 12.0, 13.5, 15.0, 16.5, 18.0, 19.5, 21.0, 22.5, 24.0, 25.5, 27.0, 28.5, 30.0, 31.5, 33.0, 34.5, 36.0, 37.5, 39.0, 40.5, 42.0, 43.5, 45.0, 46.5, 48.0, 49.5, 51.0, 52.5, 54.0, 55.5, 57.0, 58.5, 60.0, 61.5, 63.0, 64.5, 66.0, 67.5, 69.0, 70.5, 72.0, 73.5, 75.0, 76.5, 78.0, 79.5, 81.0, 82.5, 84.0, 85.5, 87.0, 88.5, 90.0, 91.5, 93.0, 94.5, 96.0, 97.5, 99.0, 100.5, 102.0, 103.5, 105.0, 106.5, 108.0, 109.5, 111.0, 112.5, 114.0, 115.5, 117.0, 118.5, 120.0, 121.5, 123.0, 124.5, 126.0, 127.5, 129.0, 130.5, 132.0, 133.5, 135.0, 136.5, 138.0, 139.5, 141.0, 142.5, 144.0, 145.5, 147.0, 148.5, 150.0];
	c: ARRAY[0..2] OF LREAL := [21.73, 73.97, 122.6];
	b: ARRAY[0..2] OF LREAL := [54.58, 118.2, 170.8];
	b_c: ARRAY[0..2] OF LREAL := [-66.3, -24.7, 15.5325443786982];
	b_d: ARRAY[0..2] OF LREAL := [4.2869822485207, 56.4869822485207, 90.1869822485207];
	e: ARRAY[0..2] OF LREAL := [73.88, 114.1, 158.0];
	b_b: ARRAY[0..2] OF SINT := [3, 3, 1];
	
	
	

END_VAR


VAR RETAIN
    nRem1 : INT :=0;
END_VAR


(* Outputs for Atomic SubSystem: '<Root>/Subsystem' *)
(* Outputs for Atomic SubSystem: '<S1>/FuzzzyCtr' *)
(* MATLAB Function: '<S2>/Evaluate Rule Antecedents' *)
(* MATLAB Function 'Evaluate Rule Antecedents': '<S4>:1' *)
(* '<S4>:1:4' if SimulateUsing==1 &amp;&amp; coder.internal.canUseExtrinsic ... *)
(* '<S4>:1:5'         &amp;&amp; (isa(inputs,'double') || isa(inputs,'single')) *)
(* '<S4>:1:32' else *)
(* '<S4>:1:33' if fis.inputFuzzySetType==1 *)
(* '<S4>:1:34' [antecedentOutputs,sumAntecedentOutputs] = ... *)
(* '<S4>:1:35'             fuzzy.internal.codegen.evaluateRuleAntecedent(... *)
(* '<S4>:1:36'             inputs,fis,diagnostics); *)
y1 := 0.0;
y2 := 0.0;

IF in >= -17.61 THEN 
    y1 := 1.0;
END_IF;


IF in < -77.61 THEN 
    y1 := 0.0;
END_IF;


IF (-77.61 <= in) AND (in < -17.61) THEN 
    y1 := (in - -77.61) * 0.016666666666666666;
END_IF;


IF in <= 4.584 THEN 
    y2 := 1.0;
END_IF;


IF in > 31.8 THEN 
    y2 := 0.0;
END_IF;


IF (4.584 < in) AND (in <= 31.8) THEN 
    y2 := (31.8 - in) * 0.036743092298647854;
END_IF;

y1 := MIN(y1, y2);
inputMFCache_idx_1 := trimf(x := in, params1 := c);
inputMFCache_idx_2 := trimf(x := in, params1 := b);

IF 1.0 <= y1 THEN 
    y1 := 1.0;
END_IF;

y2 := y1;
rtb_antecedentOutputs[0] := y1;

IF 1.0 > inputMFCache_idx_1 THEN 
    y1 := inputMFCache_idx_1;
ELSE 
    y1 := 1.0;
END_IF;

y2 := y2 + y1;
rtb_antecedentOutputs[1] := y1;

IF 1.0 > inputMFCache_idx_2 THEN 
    y1 := inputMFCache_idx_2;
ELSE 
    y1 := 1.0;
END_IF;

y2 := y2 + y1;
rtb_antecedentOutputs[2] := y1;
(* MATLAB Function: '<S2>/Evaluate Rule Consequents' incorporates:
 *  Constant: '<S2>/Output Sample Points' *)
(* MATLAB Function 'Evaluate Rule Consequents': '<S5>:1' *)
(* '<S5>:1:4' if SimulateUsing==1 &amp;&amp; coder.internal.canUseExtrinsic ... *)
(* '<S5>:1:5'         &amp;&amp; (isa(inputs,'double') || isa(inputs,'single')) *)
(* '<S5>:1:55' else *)
(* '<S5>:1:56' if fis.inputFuzzySetType==1 *)
(* '<S5>:1:57' if strcmp(char(fis.type),'mamdani') *)
(* '<S5>:1:58' aggregatedOutputs = ... *)
(* '<S5>:1:59'                 fuzzy.internal.codegen.evaluateRuleConsequentForMamdaniFIS(... *)
(* '<S5>:1:60'                 antecedentOutputs,fis,samplePoints); *)
i0_trimf_l(x := OutputSamplePoints_Value, params1 := b_c);
tmp := i0_trimf_l.y;
i0_trimf_l(x := OutputSamplePoints_Value, params1 := b_d);
tmp_0 := i0_trimf_l.y;
i0_trimf_l(x := OutputSamplePoints_Value, params1 := e);
tmp_1 := i0_trimf_l.y;
(* End of Outputs for SubSystem: '<S1>/FuzzzyCtr' *)
(* End of Outputs for SubSystem: '<Root>/Subsystem' *)
(* Outputs for Atomic SubSystem: '<Root>/Subsystem' *)
(* Outputs for Atomic SubSystem: '<S1>/FuzzzyCtr' *)
(* MATLAB Function: '<S2>/Evaluate Rule Consequents' *)

FOR ruleID := 0 TO 100 DO 
    rtb_aggregatedOutputs[ruleID] := 0.0;
    outputMFCache[3 * ruleID] := tmp[ruleID];
    outputMFCache[(3 * ruleID) + 1] := tmp_0[ruleID];
    outputMFCache[(3 * ruleID) + 2] := tmp_1[ruleID];
END_FOR;


FOR ruleID := 0 TO 2 DO 
    inputMFCache_idx_1 := rtb_antecedentOutputs[ruleID];

    FOR sampleID := 0 TO 100 DO 
        inputMFCache_idx_2 := rtb_aggregatedOutputs[sampleID];
        y1 := outputMFCache[((3 * sampleID) + SINT_TO_DINT(b_b[ruleID])) - 1];

        IF y1 > inputMFCache_idx_1 THEN 
            y1 := inputMFCache_idx_1;
        END_IF;


        IF inputMFCache_idx_2 < y1 THEN 
            inputMFCache_idx_2 := y1;
        END_IF;

        rtb_aggregatedOutputs[sampleID] := inputMFCache_idx_2;
    END_FOR;

END_FOR;

(* MATLAB Function: '<S2>/Defuzzify Outputs' incorporates:
 *  Constant: '<S2>/Output Sample Points'
 *  MATLAB Function: '<S2>/Evaluate Rule Antecedents' *)
(* MATLAB Function 'Defuzzify Outputs': '<S3>:1' *)
(* '<S3>:1:4' if SimulateUsing==1 &amp;&amp; coder.internal.canUseExtrinsic ... *)
(* '<S3>:1:5'         &amp;&amp; (isa(aggregatedOutputs,'double') || isa(aggregatedOutputs,'single')) *)
(* '<S3>:1:63' else *)
(* '<S3>:1:64' if fis.inputFuzzySetType==1 *)
(* '<S3>:1:65' if isequal(fis.type,uint8('mamdani')) *)
(* '<S3>:1:66' defuzzifiedOutputs = ... *)
(* '<S3>:1:67'                 fuzzy.internal.codegen.applyMamdaniDefuzzificationMethod(... *)
(* '<S3>:1:68'                 samplePoints,sumAntecedentOutputs,aggregatedOutputs, ... *)
(* '<S3>:1:69'                 fis,diagnostics); *)

IF y2 = 0.0 THEN 
    (* Outport: '<Root>/out' *)
    out := 75.0;
ELSE 
    y2 := 0.0;
    y1 := 0.0;

    FOR ruleID := 0 TO 100 DO 
        y1 := y1 + rtb_aggregatedOutputs[ruleID];
    END_FOR;


    IF y1 = 0.0 THEN 
        (* Outport: '<Root>/out' *)
        out := 75.0;
    ELSE 

        FOR ruleID := 0 TO 100 DO 
            y2 := (OutputSamplePoints_Value[ruleID] * rtb_aggregatedOutputs[ruleID]) + y2;
        END_FOR;

        (* Outport: '<Root>/out' incorporates:
         *  Constant: '<S2>/Output Sample Points' *)
        out := (1.0 / y1) * y2;
    END_IF;

END_IF;

out_int := LREAL_TO_INT(out);

IF in>= Qrob_control.limite_corriente THEN 
 out := 0;	
 state_aux := TRUE;
END_IF

IF state_aux THEN
	//out := 0;
	//state_aux := FALSE;
END_IF

set_move := TRUE;
IF state THEN 
	set_move := FALSE;
END_IF
	
	



nRem1 := out_int;
(* End of MATLAB Function: '<S2>/Defuzzify Outputs' *)
(* End of Outputs for SubSystem: '<S1>/FuzzzyCtr' *)
(* End of Outputs for SubSystem: '<Root>/Subsystem' *)

END_FUNCTION_BLOCK

// ---- POUs/POUs/Fuzzy/trimf_l.TcPOU
FUNCTION_BLOCK trimf_l
VAR_INPUT
	x: ARRAY[0..100] OF LREAL;
	params1: ARRAY[0..2] OF LREAL;
END_VAR
VAR_OUTPUT
	y: ARRAY[0..100] OF LREAL;
END_VAR
VAR
	a: LREAL;
	b: LREAL;
	c: LREAL;
	i: DINT;
	x_0: LREAL;
END_VAR


a := params1[0];
b := params1[1];
c := params1[2];

FOR i := 0 TO 100 DO 
    x_0 := x[i];
    y[i] := 0.0;

    IF a <> b THEN 

        IF a < x_0 THEN 

            IF x_0 < b THEN 
                y[i] := (1.0 / (b - a)) * (x_0 - a);
            END_IF;

        END_IF;

    END_IF;


    IF b <> c THEN 

        IF b < x_0 THEN 

            IF x_0 < c THEN 
                y[i] := (1.0 / (c - b)) * (c - x_0);
            END_IF;

        END_IF;

    END_IF;


    IF x_0 = b THEN 
        y[i] := 1.0;
    END_IF;

END_FOR;

END_FUNCTION_BLOCK

// ---- POUs/POUs/Fuzzy/trimf.TcPOU
FUNCTION trimf : LREAL
VAR_INPUT
	x: LREAL;
	params1: ARRAY[0..2] OF LREAL;
END_VAR
VAR
END_VAR


trimf := 0.0;

IF params1[0] <> params1[1] THEN 

    IF params1[0] < x THEN 

        IF x < params1[1] THEN 
            trimf := (1.0 / (params1[1] - params1[0])) * (x - params1[0]);
        END_IF;

    END_IF;

END_IF;


IF params1[1] <> params1[2] THEN 

    IF params1[1] < x THEN 

        IF x < params1[2] THEN 
            trimf := (1.0 / (params1[2] - params1[1])) * (params1[2] - x);
        END_IF;

    END_IF;

END_IF;


IF x = params1[1] THEN 
    trimf := 1.0;
END_IF;

END_FUNCTION

// ---- POUs/POUs/Qrob/QRob_functions/Qrob_control.TcPOU
PROGRAM Qrob_control

VAR_INPUT
	


	torque_set_point AT%Q*:INT;
	torque_enable : BOOL := FALSE;
	enable_torque_out :BOOL;
	torque_decre : REAL :=2;
	
	torque_max_vel : REAL := 200;
	
	actual_torque AT%I*:INT ;
	actual_velocity : REAL;
	done_torqte_lib : BOOL;
	t_aux : INT;
	start_plot : BOOL;
	aux_cu :REAL;
	bthome : BOOL;
	home :	 BOOL;
	reset : bool;
	external : BOOL;
    mover_horario:	BOOL;
	mover_antihorario: BOOL;
	velocidad: REAL := 10 ;
	velocidad_ext: REAL := 100 ;
	set_posicion_mover :INT := 25;
	EnableAxis1 : BOOL := TRUE;
	detener : BOOL;
	mover_abs :BOOL;
	pos_mover_abs :REAL ;
	

	
	
	ajustar_tornillo : BOOL ;
	limite_corriente : REAL := 120;
	torque_relief : BOOL := FALSE;
	tor_on : BOOL;
    tor_val : INT;
		aux_velo : BOOL;
	
END_VAR

VAR
	MC_BufferMode :MC_BufferMode;
	fbPower: MC_Power;
	Axis1Enabled : BOOL;
	actual_position : LREAL;
	//actual_velocity : REAL;
	original_vel :DINT;
	actual_current  :  LREAL;
	position_ok :BOOL;
	
	mov_abs_ok : BOOL;
	max_current : BOOL;
	val_max_current : REAL;
	aux_current : REAL;

	
	MC_Home: MC_HOME;
	MC_ReadActualPosition: MC_ReadActualPosition;
	MC_ReadActualVelocity : MC_ReadActualVelocity;
	MC_ReadParameter_0: MC_ReadParameter;
	MC_MoveVelocity_horario: MC_MoveVelocity;
	MC_MoveVelocity_antiorario: MC_MoveVelocity;
	MC_Stop: MC_Stop;
	MC_Stop2: MC_Stop;
	MC_MoveAbsolute: MC_MoveAbsolute;
    MC_TorqueControl : MC_TorqueControl;
	Ton : TON;
	RS : RS;
	limit_current : limit_current;
	
	
	fuzzy : Subsystem;
	fuzzy_vel : LREAL;
	fuzzy_active : BOOL;
	stop_limit : BOOL;
    MC_ExtSetPointGenEnable : MC_ExtSetPointGenEnable;
	MC_Reset : MC_Reset;
	MC_MoveSuperImposed : MC_MoveSuperImposed;
    FB_CTRL_SETPOINT_GENERATOR : FB_CTRL_SETPOINT_GENERATOR;

	num_ran : LREAL;
	pulse : BOOL:= TRUE;
	PT_b : BOOL;
	DRAND : DRAND;
	pulse1 : pulse_;
	nrand_out : LREAL;
   
	state_move_active : BOOL;	


Max_profile_velocity AT%Q*:UDINT := 314572;
Modes_operation AT%Q*:USINT:= 8;

END_VAR

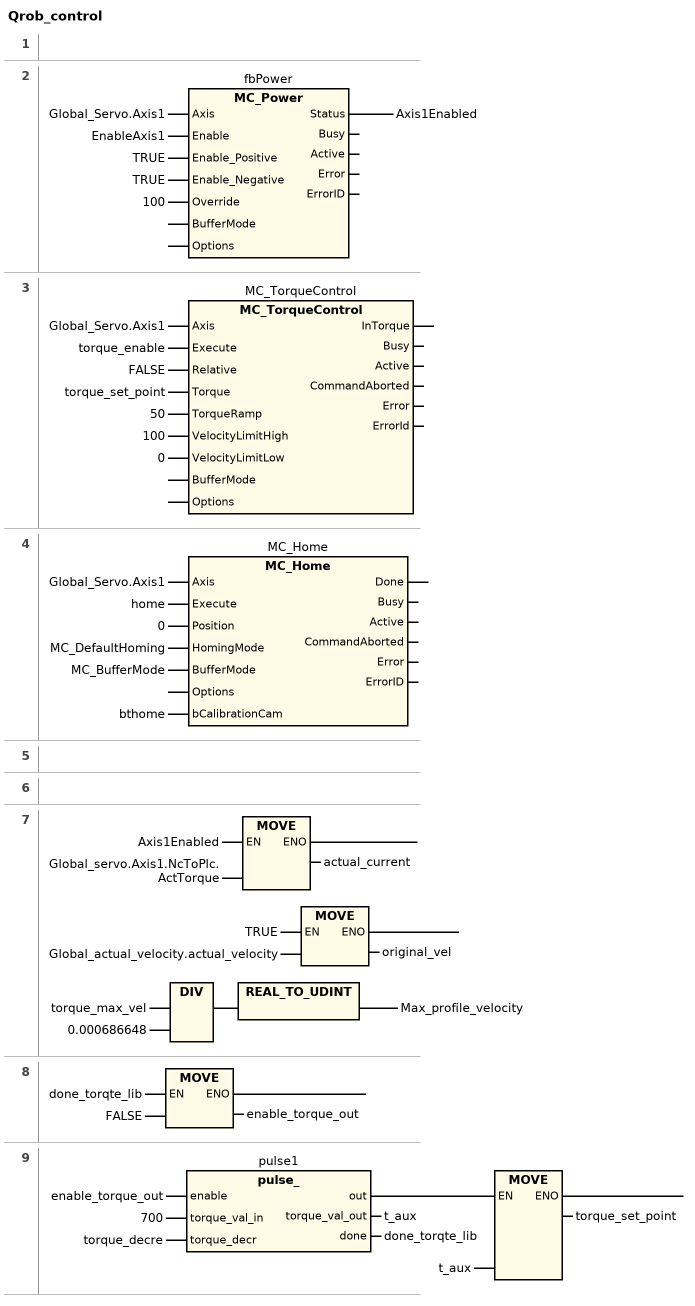
// NETWORK 1

// NETWORK 2
fbPower(
    Axis := Global_Servo.Axis1,
    Enable := EnableAxis1,
    Enable_Positive := TRUE,
    Enable_Negative := TRUE,
    Override := 100); // MC_Power
Axis1Enabled := fbPower.Status;

// NETWORK 3
MC_TorqueControl(
    Axis := Global_Servo.Axis1,
    Execute := torque_enable,
    Relative := FALSE,
    Torque := torque_set_point,
    TorqueRamp := 50,
    VelocityLimitHigh := 100,
    VelocityLimitLow := 0);

// NETWORK 4
MC_Home(
    Axis := Global_Servo.Axis1,
    Execute := home,
    Position := 0,
    HomingMode := MC_DefaultHoming,
    BufferMode := MC_BufferMode,
    bCalibrationCam := bthome);

// NETWORK 5

// NETWORK 6

// NETWORK 7
IF Axis1Enabled THEN actual_current := Global_servo.Axis1.NcToPlc.ActTorque; END_IF
original_vel := Global_actual_velocity.actual_velocity;
Max_profile_velocity := REAL_TO_UDINT(torque_max_vel / 0.000686648);

// NETWORK 8
IF done_torqte_lib THEN enable_torque_out := FALSE; END_IF

// NETWORK 9
pulse1(
    enable := enable_torque_out,
    torque_val_in := 700,
    torque_decr := torque_decre,
    torque_val_out => t_aux,
    done => done_torqte_lib); // pulse_
IF pulse1.out THEN torque_set_point := t_aux; END_IF

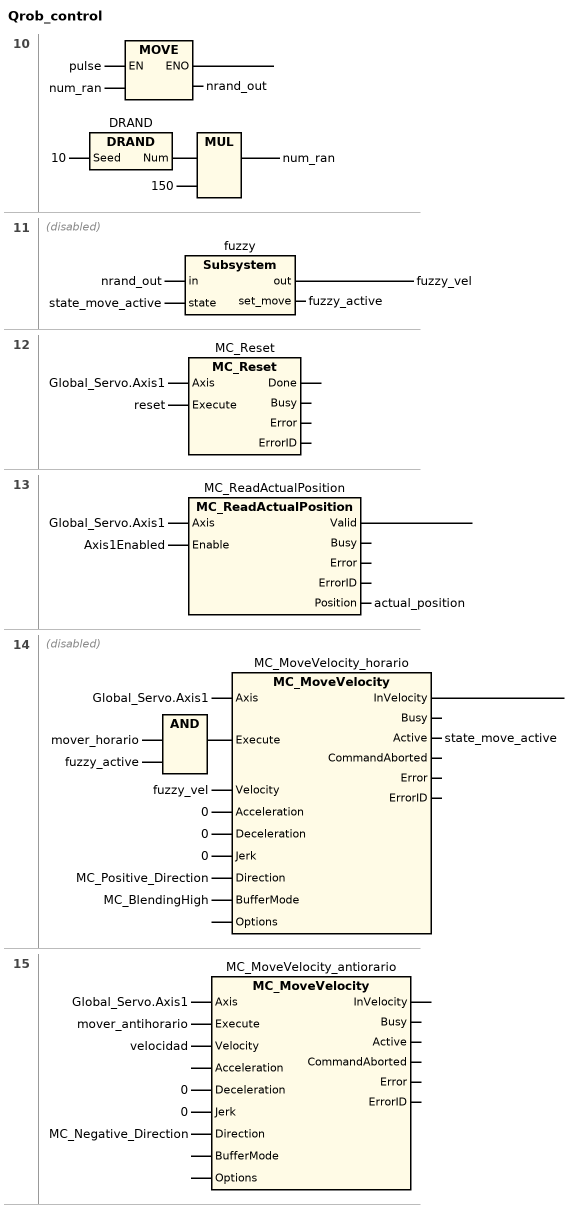
// NETWORK 10
IF pulse THEN nrand_out := num_ran; END_IF
DRAND(Seed := 10);
num_ran := DRAND.Num * 150;

// NETWORK 11 (disabled)
// fuzzy(in := nrand_out, state := state_move_active, set_move => fuzzy_active); // Subsystem
// fuzzy_vel := fuzzy.out;

// NETWORK 12
MC_Reset(Axis := Global_Servo.Axis1, Execute := reset);

// NETWORK 13
MC_ReadActualPosition(Axis := Global_Servo.Axis1, Enable := Axis1Enabled, Position => actual_position);

// NETWORK 14 (disabled)
// MC_MoveVelocity_horario(
//     Axis := Global_Servo.Axis1,
//     Execute := mover_horario AND fuzzy_active,
//     Velocity := fuzzy_vel,
//     Acceleration := 0,
//     Deceleration := 0,
//     Jerk := 0,
//     Direction := MC_Positive_Direction,
//     BufferMode := MC_BlendingHigh,
//     Active => state_move_active); // MC_MoveVelocity

// NETWORK 15
MC_MoveVelocity_antiorario(
    Axis := Global_Servo.Axis1,
    Execute := mover_antihorario,
    Velocity := velocidad,
    Deceleration := 0,
    Jerk := 0,
    Direction := MC_Negative_Direction); // MC_MoveVelocity

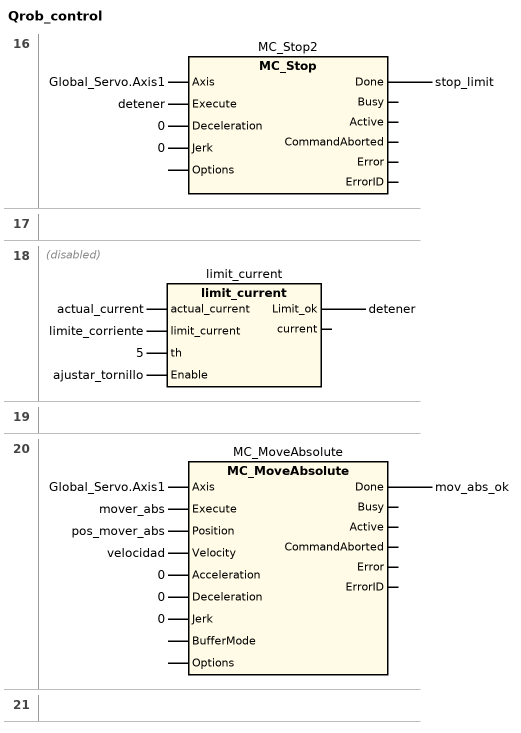
// NETWORK 16
MC_Stop2(Axis := Global_Servo.Axis1, Execute := detener, Deceleration := 0, Jerk := 0); // MC_Stop
stop_limit := MC_Stop2.Done;

// NETWORK 17

// NETWORK 18 (disabled)
// limit_current(
//     actual_current := actual_current,
//     limit_current := limite_corriente,
//     th := 5,
//     Enable := ajustar_tornillo);
// detener := limit_current.Limit_ok;

// NETWORK 19

// NETWORK 20
MC_MoveAbsolute(
    Axis := Global_Servo.Axis1,
    Execute := mover_abs,
    Position := pos_mover_abs,
    Velocity := velocidad,
    Acceleration := 0,
    Deceleration := 0,
    Jerk := 0);
mov_abs_ok := MC_MoveAbsolute.Done;

// NETWORK 21

END_PROGRAM

// ---- POUs/POUs/l/limit_current.TcPOU
FUNCTION_BLOCK limit_current
VAR_INPUT
	actual_current : REAL;
	limit_current : REAL;
	th : REAL;
	Enable : BOOL;	
	
	//relief_turn : BOOL := FALSE;	
   
	
END_VAR
VAR_OUTPUT
	Limit_ok :BOOL;
	current : REAL;
END_VAR
VAR
	A : REAL;
	B : REAL;
	
END_VAR


IF Enable = TRUE THEN 
	A := limit_current-th;
	B := limit_current +th;
	
	IF (A <= actual_current) AND (actual_current <= B) THEN 
		current := actual_current;
		IF current >= limit_current THEN
		  Limit_ok := TRUE;			 
		END_IF

	END_IF
ELSE
	 Limit_ok := FALSE;
	
END_IF

END_FUNCTION_BLOCK

// ---- POUs/POUs/l/pulse_.TcPOU
FUNCTION_BLOCK pulse_
VAR_INPUT
	enable: BOOL:= FALSE;
	torque_val_in : INT;
	torque_decr : REAL:= 2;
END_VAR
VAR_OUTPUT
	out: BOOL:= FALSE;
	torque_val_out :INT;
	done :BOOL;
	
END_VAR
VAR
	torque_aux : REAL;
END_VAR

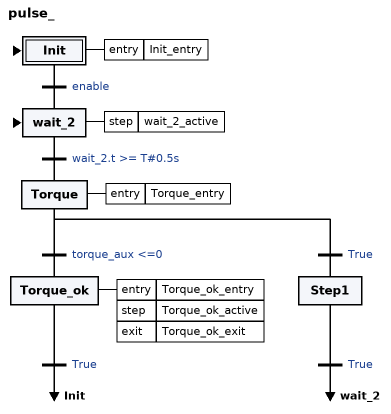
INITIAL_STEP Init:
    Init_entry(P1);  // entry action
END_STEP
TRANSITION FROM Init TO wait_2
    := enable;
END_TRANSITION
STEP wait_2:
    wait_2_active(N);  // step action
END_STEP
TRANSITION FROM wait_2 TO Torque
    := wait_2.t >= T#0.5s;
END_TRANSITION
STEP Torque:
    Torque_entry(P1);  // entry action
END_STEP
TRANSITION FROM Torque TO Torque_ok
    := torque_aux <=0;
END_TRANSITION
STEP Torque_ok:
    Torque_ok_entry(P1);  // entry action
    Torque_ok_active(N);  // step action
    Torque_ok_exit(P0);  // exit action
END_STEP
TRANSITION FROM Torque_ok TO Init
    := True;
END_TRANSITION
TRANSITION FROM Torque TO Step1
    := True;
END_TRANSITION
STEP Step1:
END_STEP
TRANSITION FROM Step1 TO wait_2
    := True;
END_TRANSITION

ACTION Init_entry:
out := FALSE;
done := False;
torque_aux := torque_val_in;
END_ACTION

ACTION Torque_entry:
torque_aux:=  ((torque_aux/torque_decr));


IF torque_aux <0 THEN
	torque_aux :=0 ;
END_IF

IF enable = TRUE THEN
torque_val_out := REAL_TO_INT(torque_aux);
END_IF
END_ACTION

ACTION Torque_ok_active:

END_ACTION

ACTION Torque_ok_entry:
out := TRUE;
done := TRue;
END_ACTION

ACTION Torque_ok_exit:
out:=FALSE;
END_ACTION

ACTION wait_1_active:
out := False;
END_ACTION

ACTION wait_2_active:
out := True;
END_ACTION

END_FUNCTION_BLOCK

// ---- POUs/POUs/IR_take_img/get_images.TcPOU
PROGRAM get_images
VAR
	start_head: BOOL;
	start_nut : BOOL;
	vi_get_img_cabezal_dere : BOOL;
	vi_get_img_nut : BOOL;
	head_ok : BOOL;
	nut_ok : BOOL;
END_VAR

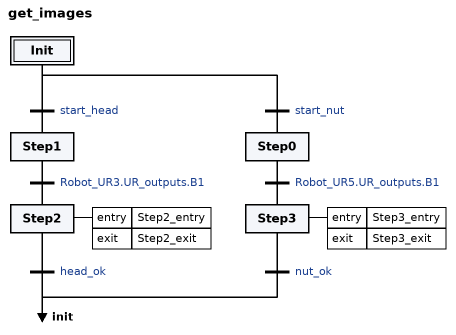
INITIAL_STEP Init:
END_STEP
TRANSITION FROM Init TO Step1
    := start_head;
END_TRANSITION
STEP Step1:
END_STEP
TRANSITION FROM Step1 TO Step2
    := Robot_UR3.UR_outputs.B1;
END_TRANSITION
STEP Step2:
    Step2_entry(P1);  // entry action
    Step2_exit(P0);  // exit action
END_STEP
TRANSITION FROM Step2 TO init
    := head_ok;
END_TRANSITION
TRANSITION FROM Init TO Step0
    := start_nut;
END_TRANSITION
STEP Step0:
END_STEP
TRANSITION FROM Step0 TO Step3
    := Robot_UR5.UR_outputs.B1;
END_TRANSITION
STEP Step3:
    Step3_entry(P1);  // entry action
    Step3_exit(P0);  // exit action
END_STEP
TRANSITION FROM Step3 TO init
    := nut_ok;
END_TRANSITION

ACTION Step2_entry:
vi_get_img_cabezal_dere := TRUE;
Robot_UR3.UR_inputs.Bits.B1 := False;
END_ACTION

ACTION Step2_exit:
vi_get_img_cabezal_dere := FALSE;
Robot_UR3.UR_inputs.Bits.B1 := TRUE;
head_ok := False;
END_ACTION

ACTION Step3_entry:
vi_get_img_nut := TRUE;
Robot_UR5.UR_inputs.Bits.B1 := False;
END_ACTION

ACTION Step3_exit:
vi_get_img_nut := FALSE;
Robot_UR5.UR_inputs.Bits.B1 := TRUE;
nut_ok := False;
END_ACTION

END_PROGRAM

// ---- POUs/POUs/l/Atornillar_ur5.TcPOU
PROGRAM Atornillar_UR5
VAR
END_VAR

VAR_INPUT
	Iniciar : Bool;
	Corriente : REAL :=10;
	Vueltas : REAL := 1;
	giro_alivio : LREAL := 0;
END_VAR
VAR_OUTPUT
END_VAR
VAR
	cal_vueltas : REAL;
	ct : INT;
	TIME_IN :TIME := T#10000MS;
	wait_t : BOOL;
END_VAR

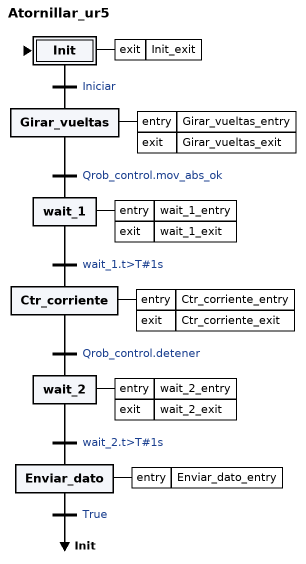
INITIAL_STEP Init:
    Init_exit(P0);  // exit action
END_STEP
TRANSITION FROM Init TO Girar_vueltas
    := Iniciar;
END_TRANSITION
STEP Girar_vueltas:
    Girar_vueltas_entry(P1);  // entry action
    Girar_vueltas_exit(P0);  // exit action
END_STEP
TRANSITION FROM Girar_vueltas TO wait_1
    := Qrob_control.mov_abs_ok;
END_TRANSITION
STEP wait_1:
    wait_1_entry(P1);  // entry action
    wait_1_exit(P0);  // exit action
END_STEP
TRANSITION FROM wait_1 TO Ctr_corriente
    := wait_1.t>T#1s;
END_TRANSITION
STEP Ctr_corriente:
    Ctr_corriente_entry(P1);  // entry action
    Ctr_corriente_exit(P0);  // exit action
END_STEP
TRANSITION FROM Ctr_corriente TO wait_2
    := Qrob_control.detener;
END_TRANSITION
STEP wait_2:
    wait_2_entry(P1);  // entry action
    wait_2_exit(P0);  // exit action
END_STEP
TRANSITION FROM wait_2 TO Enviar_dato
    := wait_2.t>T#1s;
END_TRANSITION
STEP Enviar_dato:
    Enviar_dato_entry(P1);  // entry action
END_STEP
TRANSITION FROM Enviar_dato TO Init
    := True;
END_TRANSITION

ACTION Alivio_torque_entry:
//regreo un grado para aliviar el torque y que pueda salir la herramienta
//Robot_A.UR_inputs.Bits.B11 := TRUE;
//wait_t := FALSE;
//Qrob_control.pos_mover_abs := Qrob_control.actual_position - giro_alivio;
//Qrob_control.velocidad := 50;
//Qrob_control.mover_abs := TRUE;


//Qrob_control.ajustar_tornillo := TRUE;
//Qrob_control.torque_relief := TRUE;
//Qrob_control.pos_mover_abs := Qrob_control.actual_position - giro_alivio;
//Qrob_control.velocidad := 0.5;
//Qrob_control.limite_corriente := 10;
//Qrob_control.mover_abs := TRUE;
END_ACTION

ACTION Alivio_torque_exit:

Robot_UR5.UR_inputs.Bits.B10 := FALSE;
//Qrob_control.ajustar_tornillo := FALSE;
//Qrob_control.torque_relief := FALSE;
Qrob_control.mover_abs := FALSE;
Qrob_control.detener := TRUE;
Qrob_control.detener := FALSE;
END_ACTION

ACTION Ctr_corriente_entry:
//cuando haya llegado al numero de vueltas especificado , realizo control de corriente 

wait_t := FALSE;
//FOR ct:=1 TO 5000 BY 1 DO
//Qrob_control.velocidad := 20;  
//END_FOR;

Qrob_control.ajustar_tornillo := TRUE;
Qrob_control.pos_mover_abs := 5000000;	
Qrob_control.velocidad := 100;
Qrob_control.limite_corriente := Corriente;
Qrob_control.mover_abs := TRUE;
END_ACTION

ACTION Ctr_corriente_exit:

Qrob_control.ajustar_tornillo := FALSE;
Qrob_control.detener := TRUE;
Qrob_control.detener := FALSE;
Qrob_control.mover_abs := FALSE;
END_ACTION

ACTION Enviar_dato_entry:

Robot_UR5.UR_inputs.Bits.B7 := TRUE;
Global_servo.Atornillado_ok :=TRUE;
END_ACTION

ACTION Girar_vueltas_entry:
// muevo ciertas cantidas d evuelatas a mayor velocidad y sin control de corriente 
Qrob_control.ajustar_tornillo := FALSE;


cal_vueltas := Qrob_control.actual_position + vueltas*360;
Qrob_control.pos_mover_abs := cal_vueltas;	
Qrob_control.velocidad := 180;
Qrob_control.mover_abs := TRUE;
END_ACTION

ACTION Girar_vueltas_exit:
Qrob_control.detener := TRUE;
Qrob_control.detener := FALSE;
Qrob_control.mover_abs := FALSE;
END_ACTION

ACTION Init_exit:

Robot_UR5.UR_inputs.Bits.B7 := FALSE;
Robot_UR5.UR_inputs.Bits.B8 := FALSE;
Iniciar := False;
END_ACTION

ACTION wait_1_entry:
Robot_UR5.UR_inputs.Bits.B10 := TRUE;
Qrob_control.detener := TRUE;
Qrob_control.detener := FALSE;
Qrob_control.mover_abs := FALSE;
END_ACTION

ACTION wait_1_exit:
Robot_UR5.UR_inputs.Bits.B10 := FALSE;
END_ACTION

ACTION wait_2_entry:


Qrob_control.detener := TRUE;
Qrob_control.detener := FALSE;
Qrob_control.mover_abs := FALSE;

Robot_UR5.UR_inputs.Bits.B7 := True;
END_ACTION

ACTION wait_2_exit:
Robot_UR5.UR_inputs.Bits.B7 := FALSE;
END_ACTION

END_PROGRAM

// ---- POUs/POUs/l/data_robot_ur5.TcPOU
PROGRAM data_robot_UR5
VAR
	
join_pos_1 : REAL;
join_pos_2 : REAL;
join_pos_3 : REAL;
join_pos_4 : REAL;
join_pos_5 : REAL;
join_pos_6 : REAL;

join_torque_1: REAL;
join_torque_2: REAL;
join_torque_3: REAL;
join_torque_4: REAL;
join_torque_5: REAL;
join_torque_6: REAL;

TCP_pos_x : REAL;
TCP_pos_y : REAL;
TCP_pos_z : REAL;
TCP_pos_rx : REAL;
TCP_pos_ry : REAL;
TCP_pos_rz : REAL;


TCP_force_x : REAL;
TCP_force_y : REAL;
TCP_force_z : REAL;
TCP_torque_x : REAL;
TCP_torque_y : REAL;
TCP_torque_z : REAL;

TCP_force : REAL;
velocity :INT;
turn_aux_float : REAL:= 0;
turn_aux_int : INT := 0;
qRob_actual_pos : REAL;	
new_turn : REAL;

//velocity_degress : REAL;
END_VAR


qRob_actual_pos := Get_QRob_Pos.actual_position/360;
turn_aux_int := ABS(REAL_TO_INT(qRob_actual_pos));
turn_aux_float:= turn_aux_int  - (qRob_actual_pos);
new_turn := turn_aux_float*(-1)*360;

TCP_pos_x := flip_byte(Robot_UR5.UR_TCP.FLOAT0)*1000;
TCP_pos_y := flip_byte(Robot_UR5.UR_TCP.FLOAT1)*1000;
TCP_pos_z := flip_byte(Robot_UR5.UR_TCP.FLOAT2)*1000;
TCP_pos_rx := (flip_byte(Robot_UR5.UR_TCP.FLOAT3)*180)/3.1415;
TCP_pos_ry := (flip_byte(Robot_UR5.UR_TCP.FLOAT4)*180)/3.1415;
TCP_pos_rz := (flip_byte(Robot_UR5.UR_TCP.FLOAT5)*180)/3.1415;


TCP_force  := flip_byte(Robot_UR5.UR_TCP.FLOAT18);

TCP_force_x := flip_byte(Robot_UR5.UR_TCP.FLOAT12);
TCP_force_y := flip_byte(Robot_UR5.UR_TCP.FLOAT13);
TCP_force_z := flip_byte(Robot_UR5.UR_TCP.FLOAT14);
TCP_torque_x := flip_byte(Robot_UR5.UR_TCP.FLOAT15);
TCP_torque_y := flip_byte(Robot_UR5.UR_TCP.FLOAT16);
TCP_torque_z := flip_byte(Robot_UR5.UR_TCP.FLOAT17);

join_pos_1 := (flip_byte(Robot_UR5.UR_JOINS.FLOAT0)*180)/3.1415;
join_pos_2 := (flip_byte(Robot_UR5.UR_JOINS.FLOAT1)*180)/3.1415;
join_pos_3 := (flip_byte(Robot_UR5.UR_JOINS.FLOAT2)*180)/3.1415;
join_pos_4 := (flip_byte(Robot_UR5.UR_JOINS.FLOAT3)*180)/3.1415;
join_pos_5 := (flip_byte(Robot_UR5.UR_JOINS.FLOAT4)*180)/3.1415;
join_pos_6 := (flip_byte(Robot_UR5.UR_JOINS.FLOAT5)*180)/3.1415;
 
join_torque_1 := flip_byte(Robot_UR5.UR_float_out.FLOAT0);
join_torque_2 := flip_byte(Robot_UR5.UR_float_out.FLOAT1);
join_torque_3 := flip_byte(Robot_UR5.UR_float_out.FLOAT2);
join_torque_4 := flip_byte(Robot_UR5.UR_float_out.FLOAT3);
join_torque_5 := flip_byte(Robot_UR5.UR_float_out.FLOAT4);
join_torque_6 := flip_byte(Robot_UR5.UR_float_out.FLOAT5);

END_PROGRAM

// ---- POUs/POUs/l/data_robot_ur3.TcPOU
PROGRAM data_robot_ur3





VAR
	
join_pos_1 : REAL;
join_pos_2 : REAL;
join_pos_3 : REAL;
join_pos_4 : REAL;
join_pos_5 : REAL;
join_pos_6 : REAL;

join_torque_1: REAL;
join_torque_2: REAL;
join_torque_3: REAL;
join_torque_4: REAL;
join_torque_5: REAL;
join_torque_6: REAL;

TCP_pos_x : REAL;
TCP_pos_y : REAL;
TCP_pos_z : REAL;
TCP_pos_rx : REAL;
TCP_pos_ry : REAL;
TCP_pos_rz : REAL;


TCP_force_x : REAL;
TCP_force_y : REAL;
TCP_force_z : REAL;
TCP_torque_x : REAL;
TCP_torque_y : REAL;
TCP_torque_z : REAL;

TCP_force : REAL;

END_VAR





TCP_pos_x := flip_byte(Robot_UR3.UR_TCP.FLOAT0)*1000;
TCP_pos_y := flip_byte(Robot_UR3.UR_TCP.FLOAT1)*1000;
TCP_pos_z := flip_byte(Robot_UR3.UR_TCP.FLOAT2)*1000;
TCP_pos_rx := (flip_byte(Robot_UR3.UR_TCP.FLOAT3)*180)/PI;
TCP_pos_ry := (flip_byte(Robot_UR3.UR_TCP.FLOAT4)*180)/PI;
TCP_pos_rz := (flip_byte(Robot_UR3.UR_TCP.FLOAT5)*180)/PI;


TCP_force  := flip_byte(Robot_UR3.UR_TCP.FLOAT18);

TCP_force_x := flip_byte(Robot_UR3.UR_TCP.FLOAT12);
TCP_force_y := flip_byte(Robot_UR3.UR_TCP.FLOAT13);
TCP_force_z := flip_byte(Robot_UR3.UR_TCP.FLOAT14);
TCP_torque_x := flip_byte(Robot_UR3.UR_TCP.FLOAT15);
TCP_torque_y := flip_byte(Robot_UR3.UR_TCP.FLOAT16);
TCP_torque_z := flip_byte(Robot_UR3.UR_TCP.FLOAT17);

join_pos_1 := (flip_byte(Robot_UR3.UR_JOINS.FLOAT0)*180)/PI;
join_pos_2 := (flip_byte(Robot_UR3.UR_JOINS.FLOAT1)*180)/PI;
join_pos_3 := (flip_byte(Robot_UR3.UR_JOINS.FLOAT2)*180)/PI;
join_pos_4 := (flip_byte(Robot_UR3.UR_JOINS.FLOAT3)*180)/PI;
join_pos_5 := (flip_byte(Robot_UR3.UR_JOINS.FLOAT4)*180)/PI;
join_pos_6 := (flip_byte(Robot_UR3.UR_JOINS.FLOAT5)*180)/PI;
 
join_torque_1 := flip_byte(Robot_UR3.UR_float_out.FLOAT0);
join_torque_2 := flip_byte(Robot_UR3.UR_float_out.FLOAT1);
join_torque_3 := flip_byte(Robot_UR3.UR_float_out.FLOAT2);
join_torque_4 := flip_byte(Robot_UR3.UR_float_out.FLOAT3);
join_torque_5 := flip_byte(Robot_UR3.UR_float_out.FLOAT4);
join_torque_6 := flip_byte(Robot_UR3.UR_float_out.FLOAT5);

END_PROGRAM

// ---- POUs/POUs/miscellaneous/POU.TcPOU
PROGRAM POU
VAR
END_VAR

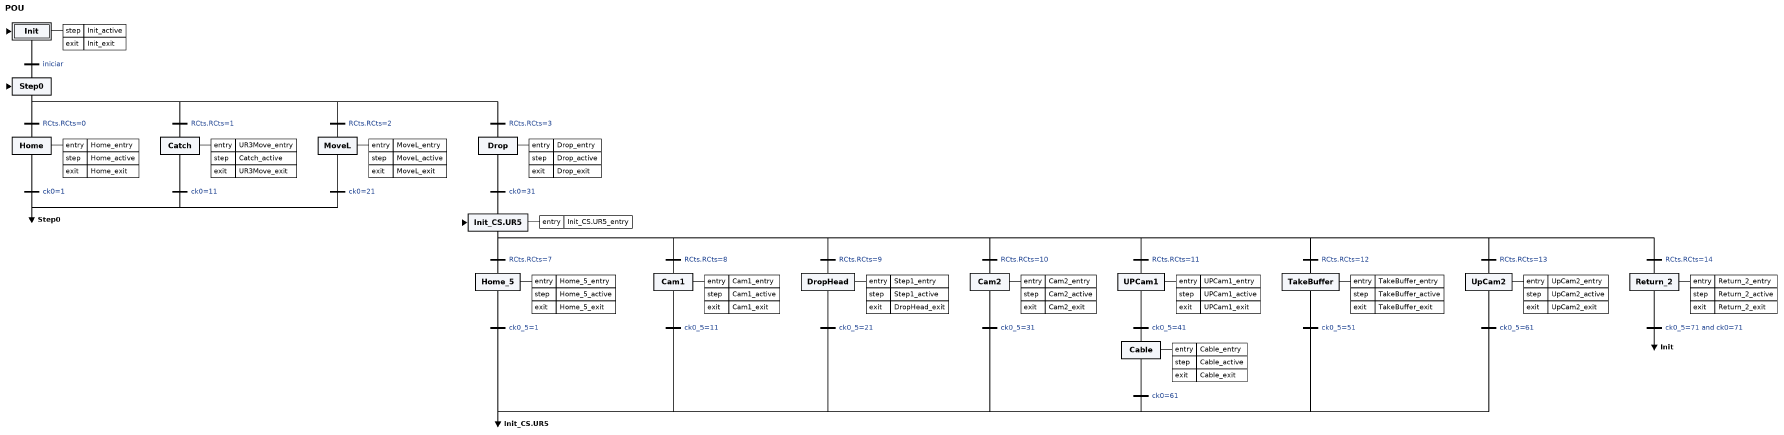
INITIAL_STEP Init:
    Init_active(N);  // step action
    Init_exit(P0);  // exit action
END_STEP
TRANSITION FROM Init TO Step0
    := iniciar;
END_TRANSITION
STEP Step0:
END_STEP
TRANSITION FROM Step0 TO Home
    := RCts.RCts=0;
END_TRANSITION
STEP Home:
    Home_entry(P1);  // entry action
    Home_active(N);  // step action
    Home_exit(P0);  // exit action
END_STEP
TRANSITION FROM Home TO Step0
    := ck0=1;
END_TRANSITION
TRANSITION FROM Step0 TO Catch
    := RCts.RCts=1;
END_TRANSITION
STEP Catch:
    UR3Move_entry(P1);  // entry action
    Catch_active(N);  // step action
    UR3Move_exit(P0);  // exit action
END_STEP
TRANSITION FROM Catch TO Step0
    := ck0=11;
END_TRANSITION
TRANSITION FROM Step0 TO MoveL
    := RCts.RCts=2;
END_TRANSITION
STEP MoveL:
    MoveL_entry(P1);  // entry action
    MoveL_active(N);  // step action
    MoveL_exit(P0);  // exit action
END_STEP
TRANSITION FROM MoveL TO Step0
    := ck0=21;
END_TRANSITION
TRANSITION FROM Step0 TO Drop
    := RCts.RCts=3;
END_TRANSITION
STEP Drop:
    Drop_entry(P1);  // entry action
    Drop_active(N);  // step action
    Drop_exit(P0);  // exit action
END_STEP
TRANSITION FROM Drop TO Init_CS_UR5
    := ck0=31;
END_TRANSITION
STEP Init_CS_UR5:  // name as stored: Init_CS.UR5
    Init_CS.UR5_entry(P1);  // entry action
END_STEP
TRANSITION FROM Init_CS_UR5 TO Home_5
    := RCts.RCts=7;
END_TRANSITION
STEP Home_5:
    Home_5_entry(P1);  // entry action
    Home_5_active(N);  // step action
    Home_5_exit(P0);  // exit action
END_STEP
TRANSITION FROM Home_5 TO Init_CS_UR5
    := ck0_5=1;
END_TRANSITION
TRANSITION FROM Init_CS_UR5 TO Cam1
    := RCts.RCts=8;
END_TRANSITION
STEP Cam1:
    Cam1_entry(P1);  // entry action
    Cam1_active(N);  // step action
    Cam1_exit(P0);  // exit action
END_STEP
TRANSITION FROM Cam1 TO Init_CS_UR5
    := ck0_5=11;
END_TRANSITION
TRANSITION FROM Init_CS_UR5 TO DropHead
    := RCts.RCts=9;
END_TRANSITION
STEP DropHead:
    Step1_entry(P1);  // entry action
    Step1_active(N);  // step action
    DropHead_exit(P0);  // exit action
END_STEP
TRANSITION FROM DropHead TO Init_CS_UR5
    := ck0_5=21;
END_TRANSITION
TRANSITION FROM Init_CS_UR5 TO Cam2
    := RCts.RCts=10;
END_TRANSITION
STEP Cam2:
    Cam2_entry(P1);  // entry action
    Cam2_active(N);  // step action
    Cam2_exit(P0);  // exit action
END_STEP
TRANSITION FROM Cam2 TO Init_CS_UR5
    := ck0_5=31;
END_TRANSITION
TRANSITION FROM Init_CS_UR5 TO UPCam1
    := RCts.RCts=11;
END_TRANSITION
STEP UPCam1:
    UPCam1_entry(P1);  // entry action
    UPCam1_active(N);  // step action
    UPCam1_exit(P0);  // exit action
END_STEP
TRANSITION FROM UPCam1 TO Cable
    := ck0_5=41;
END_TRANSITION
STEP Cable:
    Cable_entry(P1);  // entry action
    Cable_active(N);  // step action
    Cable_exit(P0);  // exit action
END_STEP
TRANSITION FROM Cable TO Init_CS_UR5
    := ck0=61;
END_TRANSITION
TRANSITION FROM Init_CS_UR5 TO TakeBuffer
    := RCts.RCts=12;
END_TRANSITION
STEP TakeBuffer:
    TakeBuffer_entry(P1);  // entry action
    TakeBuffer_active(N);  // step action
    TakeBuffer_exit(P0);  // exit action
END_STEP
TRANSITION FROM TakeBuffer TO Init_CS_UR5
    := ck0_5=51;
END_TRANSITION
TRANSITION FROM Init_CS_UR5 TO UpCam2
    := RCts.RCts=13;
END_TRANSITION
STEP UpCam2:
    UpCam2_entry(P1);  // entry action
    UpCam2_active(N);  // step action
    UpCam2_exit(P0);  // exit action
END_STEP
TRANSITION FROM UpCam2 TO Init_CS_UR5
    := ck0_5=61;
END_TRANSITION
TRANSITION FROM Init_CS_UR5 TO Return_2
    := RCts.RCts=14;
END_TRANSITION
STEP Return_2:
    Return_2_entry(P1);  // entry action
    Return_2_active(N);  // step action
    Return_2_exit(P0);  // exit action
END_STEP
TRANSITION FROM Return_2 TO Init
    := ck0_5=71 and ck0=71;
END_TRANSITION

END_PROGRAM

// ---- POUs/POUs/miscellaneous/profinet_UR3.TcPOU
PROGRAM profinet_UR3
VAR
END_VAR

VAR_INPUT
	state : INT:=-1;
	state0 : INT:= -1; 
	state1 : INT:= -1;
	state2 : INT:= -1;
	ck0 : INT;
	ck1 : INT;
	ck2 : INT;
END_VAR


//escribir del plc al robot 
Robot_UR3.UR_inputs.Ints.INT0 := flip_int(state0);
Robot_UR3.UR_inputs.Ints.INT1 := flip_int(state1);
Robot_UR3.UR_inputs.Ints.INT2 := flip_int(state2);

//leer del robot al plc
ck0 := flip_byte_int(Robot_UR3.UR_outputs_int.INT3);
ck1 := flip_byte_int(Robot_UR3.UR_outputs_int.INT4);
ck2 := flip_byte_int(Robot_UR3.UR_outputs_int.INT5);

state0:=state;
state1:=state;
state2:=state;

IF (ck0=301 AND ck1=301 AND ck2=301) OR (ck0<>301 AND ck1=301 AND ck2=301) OR (ck0=301 AND ck1<>301 AND ck2=301) OR (ck0=301 AND ck1=301 AND ck2<>301) THEN
state:=-1;
state0 := -1;
state1 := -1;
state2 := -1;
Robot_UR3.UR_inputs.Ints.INT0 := flip_int(state0);
Robot_UR3.UR_inputs.Ints.INT1 := flip_int(state1);
Robot_UR3.UR_inputs.Ints.INT2 := flip_int(state2);
ELSIF (ck0=311 AND ck1=311 AND ck2=311) OR (ck0<>311 AND ck1=311 AND ck2=311) OR (ck0=311 AND ck1<>311 AND ck2=311) OR (ck0=311 AND ck1=311 AND ck2<>311) THEN
state:=-1;	
state0 := -1;
state1 := -1;
state2 := -1;
Robot_UR3.UR_inputs.Ints.INT0 := flip_int(state0);
Robot_UR3.UR_inputs.Ints.INT1 := flip_int(state1);
Robot_UR3.UR_inputs.Ints.INT2 := flip_int(state2);
ELSIF (ck0=321 AND ck1=321 AND ck2=321) OR (ck0<>321 AND ck1=321 AND ck2=321) OR (ck0=321 AND ck1<>321 AND ck2=321) OR (ck0=321 AND ck1=321 AND ck2<>321) THEN
state:=-1;	
state0 := -1;
state1 := -1;
state2 := -1;
Robot_UR3.UR_inputs.Ints.INT0 := flip_int(state0);
Robot_UR3.UR_inputs.Ints.INT1 := flip_int(state1);
Robot_UR3.UR_inputs.Ints.INT2 := flip_int(state2);
ELSIF (ck0=331 AND ck1=331 AND ck2=331) OR (ck0<>331 AND ck1=331 AND ck2=331) OR (ck0=331 AND ck1<>331 AND ck2=331) OR (ck0=331 AND ck1=331 AND ck2<>331) THEN
state:=-1;	
state0 := -1;
state1 := -1;
state2 := -1;
Robot_UR3.UR_inputs.Ints.INT0 := flip_int(state0);
Robot_UR3.UR_inputs.Ints.INT1 := flip_int(state1);
Robot_UR3.UR_inputs.Ints.INT2 := flip_int(state2);
ELSIF (ck0=341 AND ck1=341 AND ck2=341) OR (ck0<>341 AND ck1=341 AND ck2=341) OR (ck0=341 AND ck1<>341 AND ck2=341) OR (ck0=341 AND ck1=341 AND ck2<>341) THEN
state:=-1;	
state0 := -1;
state1 := -1;
state2 := -1;
Robot_UR3.UR_inputs.Ints.INT0 := flip_int(state0);
Robot_UR3.UR_inputs.Ints.INT1 := flip_int(state1);
Robot_UR3.UR_inputs.Ints.INT2 := flip_int(state2);
ELSIF (ck0=351 AND ck1=351 AND ck2=351) OR (ck0<>351 AND ck1=351 AND ck2=351) OR (ck0=351 AND ck1<>351 AND ck2=351) OR (ck0=351 AND ck1=351 AND ck2<>351) THEN
state:=-1;	
state0 := -1;
state1 := -1;
state2 := -1;
Robot_UR3.UR_inputs.Ints.INT0 := flip_int(state0);
Robot_UR3.UR_inputs.Ints.INT1 := flip_int(state1);
Robot_UR3.UR_inputs.Ints.INT2 := flip_int(state2);
ELSIF (ck0=361 AND ck1=361 AND ck2=361) OR (ck0<>361 AND ck1=361 AND ck2=361) OR (ck0=361 AND ck1<>361 AND ck2=361) OR (ck0=361 AND ck1=361 AND ck2<>361) THEN
state:=-1;	
state0 := -1;
state1 := -1;
state2 := -1;
Robot_UR3.UR_inputs.Ints.INT0 := flip_int(state0);
Robot_UR3.UR_inputs.Ints.INT1 := flip_int(state1);
Robot_UR3.UR_inputs.Ints.INT2 := flip_int(state2);
ELSIF (ck0=371 AND ck1=371 AND ck2=371) OR (ck0<>371 AND ck1=371 AND ck2=371) OR (ck0=371 AND ck1<>371 AND ck2=371) OR (ck0=371 AND ck1=371 AND ck2<>371) THEN
state:=-1;
state0 := -1;
state1 := -1;
state2 := -1;
Robot_UR3.UR_inputs.Ints.INT0 := flip_int(state0);
Robot_UR3.UR_inputs.Ints.INT1 := flip_int(state1);
Robot_UR3.UR_inputs.Ints.INT2 := flip_int(state2);	
END_IF

END_PROGRAM

// ---- POUs/POUs/miscellaneous/profinet_UR5.TcPOU
PROGRAM profinet_CS.UR5
VAR
END_VAR

VAR_INPUT
	state : INT:=-1;
	state0 : INT:= -1; 
	state1 : INT:= -1;
	state2 : INT:= -1;
	ck0 : INT;
	ck1 : INT;
	ck2 : INT;
END_VAR


//escribir del plc al robot 
Robot_UR5.UR_inputs.Ints.INT0 := flip_int(state0);
Robot_UR5.UR_inputs.Ints.INT1 := flip_int(state1);
Robot_UR5.UR_inputs.Ints.INT2 := flip_int(state2);

//leer del robot al plc
ck0 := flip_byte_int(Robot_UR5.UR_outputs_int.INT3);
ck1 := flip_byte_int(Robot_UR5.UR_outputs_int.INT4);
ck2 := flip_byte_int(Robot_UR5.UR_outputs_int.INT5);

state0:=state;
state1:=state;
state2:=state;

IF (ck0=501 AND ck1=501 AND ck2=501) OR (ck0<>501 AND ck1=501 AND ck2=501) OR (ck0=501 AND ck1<>501 AND ck2=501) OR (ck0=501 AND ck1=501 AND ck2<>501) THEN
state:=-1;
state0 := -1;
state1 := -1;
state2 := -1;
Robot_UR5.UR_inputs.Ints.INT0 := flip_int(state0);
Robot_UR5.UR_inputs.Ints.INT1 := flip_int(state1);
Robot_UR5.UR_inputs.Ints.INT2 := flip_int(state2);
ELSIF (ck0=511 AND ck1=511 AND ck2=511) OR (ck0<>511 AND ck1=511 AND ck2=511) OR (ck0=511 AND ck1<>511 AND ck2=511) OR (ck0=511 AND ck1=511 AND ck2<>511) THEN
state:=-1;	
state0 := -1;
state1 := -1;
state2 := -1;
Robot_UR5.UR_inputs.Ints.INT0 := flip_int(state0);
Robot_UR5.UR_inputs.Ints.INT1 := flip_int(state1);
Robot_UR5.UR_inputs.Ints.INT2 := flip_int(state2);
ELSIF (ck0=521 AND ck1=521 AND ck2=521) OR (ck0<>521 AND ck1=521 AND ck2=521) OR (ck0=521 AND ck1<>521 AND ck2=521) OR (ck0=521 AND ck1=521 AND ck2<>521) THEN
state:=-1;	
state0 := -1;
state1 := -1;
state2 := -1;
Robot_UR5.UR_inputs.Ints.INT0 := flip_int(state0);
Robot_UR5.UR_inputs.Ints.INT1 := flip_int(state1);
Robot_UR5.UR_inputs.Ints.INT2 := flip_int(state2);
ELSIF (ck0=531 AND ck1=531 AND ck2=531) OR (ck0<>531 AND ck1=531 AND ck2=531) OR (ck0=531 AND ck1<>531 AND ck2=531) OR (ck0=531 AND ck1=531 AND ck2<>531) THEN
state:=-1;	
state0 := -1;
state1 := -1;
state2 := -1;
Robot_UR5.UR_inputs.Ints.INT0 := flip_int(state0);
Robot_UR5.UR_inputs.Ints.INT1 := flip_int(state1);
Robot_UR5.UR_inputs.Ints.INT2 := flip_int(state2);
ELSIF (ck0=541 AND ck1=541 AND ck2=541) OR (ck0<>541 AND ck1=541 AND ck2=541) OR (ck0=541 AND ck1<>541 AND ck2=541) OR (ck0=541 AND ck1=541 AND ck2<>541) THEN
state:=-1;	
state0 := -1;
state1 := -1;
state2 := -1;
Robot_UR5.UR_inputs.Ints.INT0 := flip_int(state0);
Robot_UR5.UR_inputs.Ints.INT1 := flip_int(state1);
Robot_UR5.UR_inputs.Ints.INT2 := flip_int(state2);
ELSIF (ck0=551 AND ck1=551 AND ck2=551) OR (ck0<>551 AND ck1=551 AND ck2=551) OR (ck0=551 AND ck1<>551 AND ck2=551) OR (ck0=551 AND ck1=551 AND ck2<>551) THEN
state:=-1;	
state0 := -1;
state1 := -1;
state2 := -1;
Robot_UR5.UR_inputs.Ints.INT0 := flip_int(state0);
Robot_UR5.UR_inputs.Ints.INT1 := flip_int(state1);
Robot_UR5.UR_inputs.Ints.INT2 := flip_int(state2);
ELSIF (ck0=561 AND ck1=561 AND ck2=561) OR (ck0<>561 AND ck1=561 AND ck2=561) OR (ck0=561 AND ck1<>561 AND ck2=561) OR (ck0=561 AND ck1=561 AND ck2<>561) THEN
state:=-1;	
state0 := -1;
state1 := -1;
state2 := -1;
Robot_UR5.UR_inputs.Ints.INT0 := flip_int(state0);
Robot_UR5.UR_inputs.Ints.INT1 := flip_int(state1);
Robot_UR5.UR_inputs.Ints.INT2 := flip_int(state2);
ELSIF (ck0=571 AND ck1=571 AND ck2=571) OR (ck0<>571 AND ck1=571 AND ck2=571) OR (ck0=571 AND ck1<>571 AND ck2=571) OR (ck0=571 AND ck1=571 AND ck2<>571) THEN
state:=-1;
state0 := -1;
state1 := -1;
state2 := -1;
Robot_UR5.UR_inputs.Ints.INT0 := flip_int(state0);
Robot_UR5.UR_inputs.Ints.INT1 := flip_int(state1);
Robot_UR5.UR_inputs.Ints.INT2 := flip_int(state2);
ELSIF (ck0=581 AND ck1=581 AND ck2=581) OR (ck0<>581 AND ck1=581 AND ck2=581) OR (ck0=581 AND ck1<>581 AND ck2=581) OR (ck0=581 AND ck1=581 AND ck2<>581) THEN
state:=-1;
state0 := -1;
state1 := -1;
state2 := -1;
Robot_UR5.UR_inputs.Ints.INT0 := flip_int(state0);
Robot_UR5.UR_inputs.Ints.INT1 := flip_int(state1);
Robot_UR5.UR_inputs.Ints.INT2 := flip_int(state2);
ELSIF (ck0=591 AND ck1=591 AND ck2=591) OR (ck0<>591 AND ck1=591 AND ck2=591) OR (ck0=591 AND ck1<>591 AND ck2=591) OR (ck0=591 AND ck1=591 AND ck2<>591) THEN
state:=-1;
state0 := -1;
state1 := -1;
state2 := -1;
Robot_UR5.UR_inputs.Ints.INT0 := flip_int(state0);
Robot_UR5.UR_inputs.Ints.INT1 := flip_int(state1);
Robot_UR5.UR_inputs.Ints.INT2 := flip_int(state2);
ELSIF (ck0=5101 AND ck1=5101 AND ck2=5101) OR (ck0<>5101 AND ck1=5101 AND ck2=5101) OR (ck0=5101 AND ck1<>5101 AND ck2=5101) OR (ck0=5101 AND ck1=5101 AND ck2<>5101) THEN
state:=-1;
state0 := -1;
state1 := -1;
state2 := -1;
Robot_UR5.UR_inputs.Ints.INT0 := flip_int(state0);
Robot_UR5.UR_inputs.Ints.INT1 := flip_int(state1);
Robot_UR5.UR_inputs.Ints.INT2 := flip_int(state2);
ELSIF (ck0=5111 AND ck1=5111 AND ck2=5111) OR (ck0<>5111 AND ck1=5111 AND ck2=5111) OR (ck0=5111 AND ck1<>5111 AND ck2=5111) OR (ck0=5111 AND ck1=5111 AND ck2<>5111) THEN
state:=-1;
state0 := -1;
state1 := -1;
state2 := -1;
Robot_UR5.UR_inputs.Ints.INT0 := flip_int(state0);
Robot_UR5.UR_inputs.Ints.INT1 := flip_int(state1);
Robot_UR5.UR_inputs.Ints.INT2 := flip_int(state2);
ELSIF (ck0=5121 AND ck1=5121 AND ck2=5121) OR (ck0<>5121 AND ck1=5121 AND ck2=5121) OR (ck0=5121 AND ck1<>5121 AND ck2=5121) OR (ck0=5121 AND ck1=5121 AND ck2<>5121) THEN
state:=-1;
state0 := -1;
state1 := -1;
state2 := -1;
Robot_UR5.UR_inputs.Ints.INT0 := flip_int(state0);
Robot_UR5.UR_inputs.Ints.INT1 := flip_int(state1);
Robot_UR5.UR_inputs.Ints.INT2 := flip_int(state2);	
END_IF

END_PROGRAM

// ---- POUs/POUs/miscellaneous/UR3_Robot.TcPOU
PROGRAM UR3_Robot
VAR
	iniciar_secuencia_1 : BOOL;

	pos_separator_ok : BOOL;
	vi_get_img : BOOL ;
	estado_cabezal :INT;
	cabezal :BOOL;
	vi_img_ok : BOOL;
	i : BOOL;
	
	giro_cabezal :REAL;

	cx : REAL;
	cy : REAL;
	turn : REAL;
	cabezal_retirado :BOOL;
	regresar : BOOL;
	vi_image_proces: BOOL; 
	poner_cabeza : BOOL;
	
	vi_img_cabezal_dere_ok : BOOL;
	vi_img_cabezal_dere_proc_ok : BOOL;
	vi_get_img_cabezal_dere : BOOL;


END_VAR

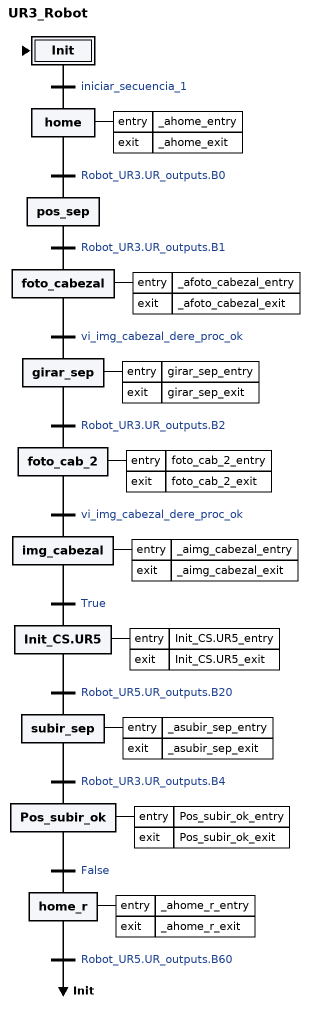
INITIAL_STEP Init:
END_STEP
TRANSITION FROM Init TO home
    := iniciar_secuencia_1;
END_TRANSITION
STEP home:
    _ahome_entry(P1);  // entry action
    _ahome_exit(P0);  // exit action
END_STEP
TRANSITION FROM home TO pos_sep
    := Robot_UR3.UR_outputs.B0;
END_TRANSITION
STEP pos_sep:
END_STEP
TRANSITION FROM pos_sep TO foto_cabezal
    := Robot_UR3.UR_outputs.B1;
END_TRANSITION
STEP foto_cabezal:
    _afoto_cabezal_entry(P1);  // entry action
    _afoto_cabezal_exit(P0);  // exit action
END_STEP
TRANSITION FROM foto_cabezal TO girar_sep
    := vi_img_cabezal_dere_proc_ok;
END_TRANSITION
STEP girar_sep:
    girar_sep_entry(P1);  // entry action
    girar_sep_exit(P0);  // exit action
END_STEP
TRANSITION FROM girar_sep TO foto_cab_2
    := Robot_UR3.UR_outputs.B2;
END_TRANSITION
STEP foto_cab_2:
    foto_cab_2_entry(P1);  // entry action
    foto_cab_2_exit(P0);  // exit action
END_STEP
TRANSITION FROM foto_cab_2 TO img_cabezal
    := vi_img_cabezal_dere_proc_ok;
END_TRANSITION
STEP img_cabezal:
    _aimg_cabezal_entry(P1);  // entry action
    _aimg_cabezal_exit(P0);  // exit action
END_STEP
TRANSITION FROM img_cabezal TO Init_CS_UR5
    := True;
END_TRANSITION
STEP Init_CS_UR5:  // name as stored: Init_CS.UR5
    Init_CS.UR5_entry(P1);  // entry action
    Init_CS.UR5_exit(P0);  // exit action
END_STEP
TRANSITION FROM Init_CS_UR5 TO subir_sep
    := Robot_UR5.UR_outputs.B20;
END_TRANSITION
STEP subir_sep:
    _asubir_sep_entry(P1);  // entry action
    _asubir_sep_exit(P0);  // exit action
END_STEP
TRANSITION FROM subir_sep TO Pos_subir_ok
    := Robot_UR3.UR_outputs.B4;
END_TRANSITION
STEP Pos_subir_ok:
    Pos_subir_ok_entry(P1);  // entry action
    Pos_subir_ok_exit(P0);  // exit action
END_STEP
TRANSITION FROM Pos_subir_ok TO home_r
    := False;
END_TRANSITION
STEP home_r:
    _ahome_r_entry(P1);  // entry action
    _ahome_r_exit(P0);  // exit action
END_STEP
TRANSITION FROM home_r TO Init
    := Robot_UR5.UR_outputs.B60;
END_TRANSITION

ACTION _afoto_cabezal_entry:
vi_get_img_cabezal_dere := TRUE;
END_ACTION

ACTION _afoto_cabezal_exit:
vi_get_img_cabezal_dere := FALSE;
vi_img_cabezal_dere_proc_ok := FALSE;
data_to_robot.head_roll_left := turn;
END_ACTION

ACTION _ahome_entry:
Robot_UR3.UR_inputs.Bits.B0 := TRUE;
END_ACTION

ACTION _ahome_exit:
Robot_UR3.UR_inputs.Bits.B0 := False;
END_ACTION

ACTION _ahome_r_entry:
Robot_UR5.UR_inputs.Bits.B27 := TRUE;
regresar := False;
END_ACTION

ACTION _ahome_r_exit:
Robot_UR5.UR_inputs.Bits.B27 := False;
END_ACTION

ACTION _aimg_cabezal_entry:
pos_separator_ok := TRUE;
END_ACTION

ACTION _aimg_cabezal_exit:
pos_separator_ok := False;
END_ACTION

ACTION _asubir_sep_entry:
Robot_UR3.UR_inputs.Bits.B20 := TRUE;
END_ACTION

ACTION _asubir_sep_exit:
Robot_UR3.UR_inputs.Bits.B20 := FALSE;
END_ACTION

ACTION foto_cab_2_entry:
vi_get_img_cabezal_dere := TRUE;
END_ACTION

ACTION foto_cab_2_exit:
vi_get_img_cabezal_dere := FALSE;
vi_img_cabezal_dere_proc_ok := FALSE;
data_to_robot.head_roll_right := turn;
END_ACTION

ACTION girar_sep_entry:
Robot_UR3.UR_inputs.Bits.B0 := TRUE;
END_ACTION

ACTION girar_sep_exit:
Robot_UR3.UR_inputs.Bits.B0 := False;
END_ACTION

ACTION Init_UR5_entry:
RCts.RCts.UR5_robot.iniciar := True;
END_ACTION

ACTION Init_UR5_exit:
RCts.RCts.UR5_robot.iniciar := False;
END_ACTION

ACTION Pos_subir_ok_entry:
Robot_UR5.UR_inputs.Bits.B20 := TRUE;
END_ACTION

ACTION Pos_subir_ok_exit:
Robot_UR5.UR_inputs.Bits.B20 := False;
END_ACTION

END_PROGRAM

// ---- POUs/POUs/miscellaneous/UR5_robot.TcPOU
PROGRAM UR5_robot
VAR
//banderas



i : BOOL := FALSE;
i2 : BOOL := FALSE;

vi_get_img : BOOL;
vi_img_ok: BOOL;

cx : REAL;
cy : REAL;
giro : REAL;
centro_ok : BOOL;
motor_pos_ok : BOOL;


// variables cabezal
giro_cabezal_dere : REAL;

vi_img_cabezal_dere_ok : BOOL;
vi_img_cabezal_dere_proc_ok : BOOL;
vi_get_img_cabezal_dere : BOOL;
vi_get_img_tuerca : BOOL;
giro_desartonillado : REAL;
cal_vueltas : REAL;
giro_aux_int : DINT;
giro_aux_float : REAL;

Atornillar: INT;
END_VAR

VAR_INPUT	
iniciar: BOOL := FALSE;
END_VAR

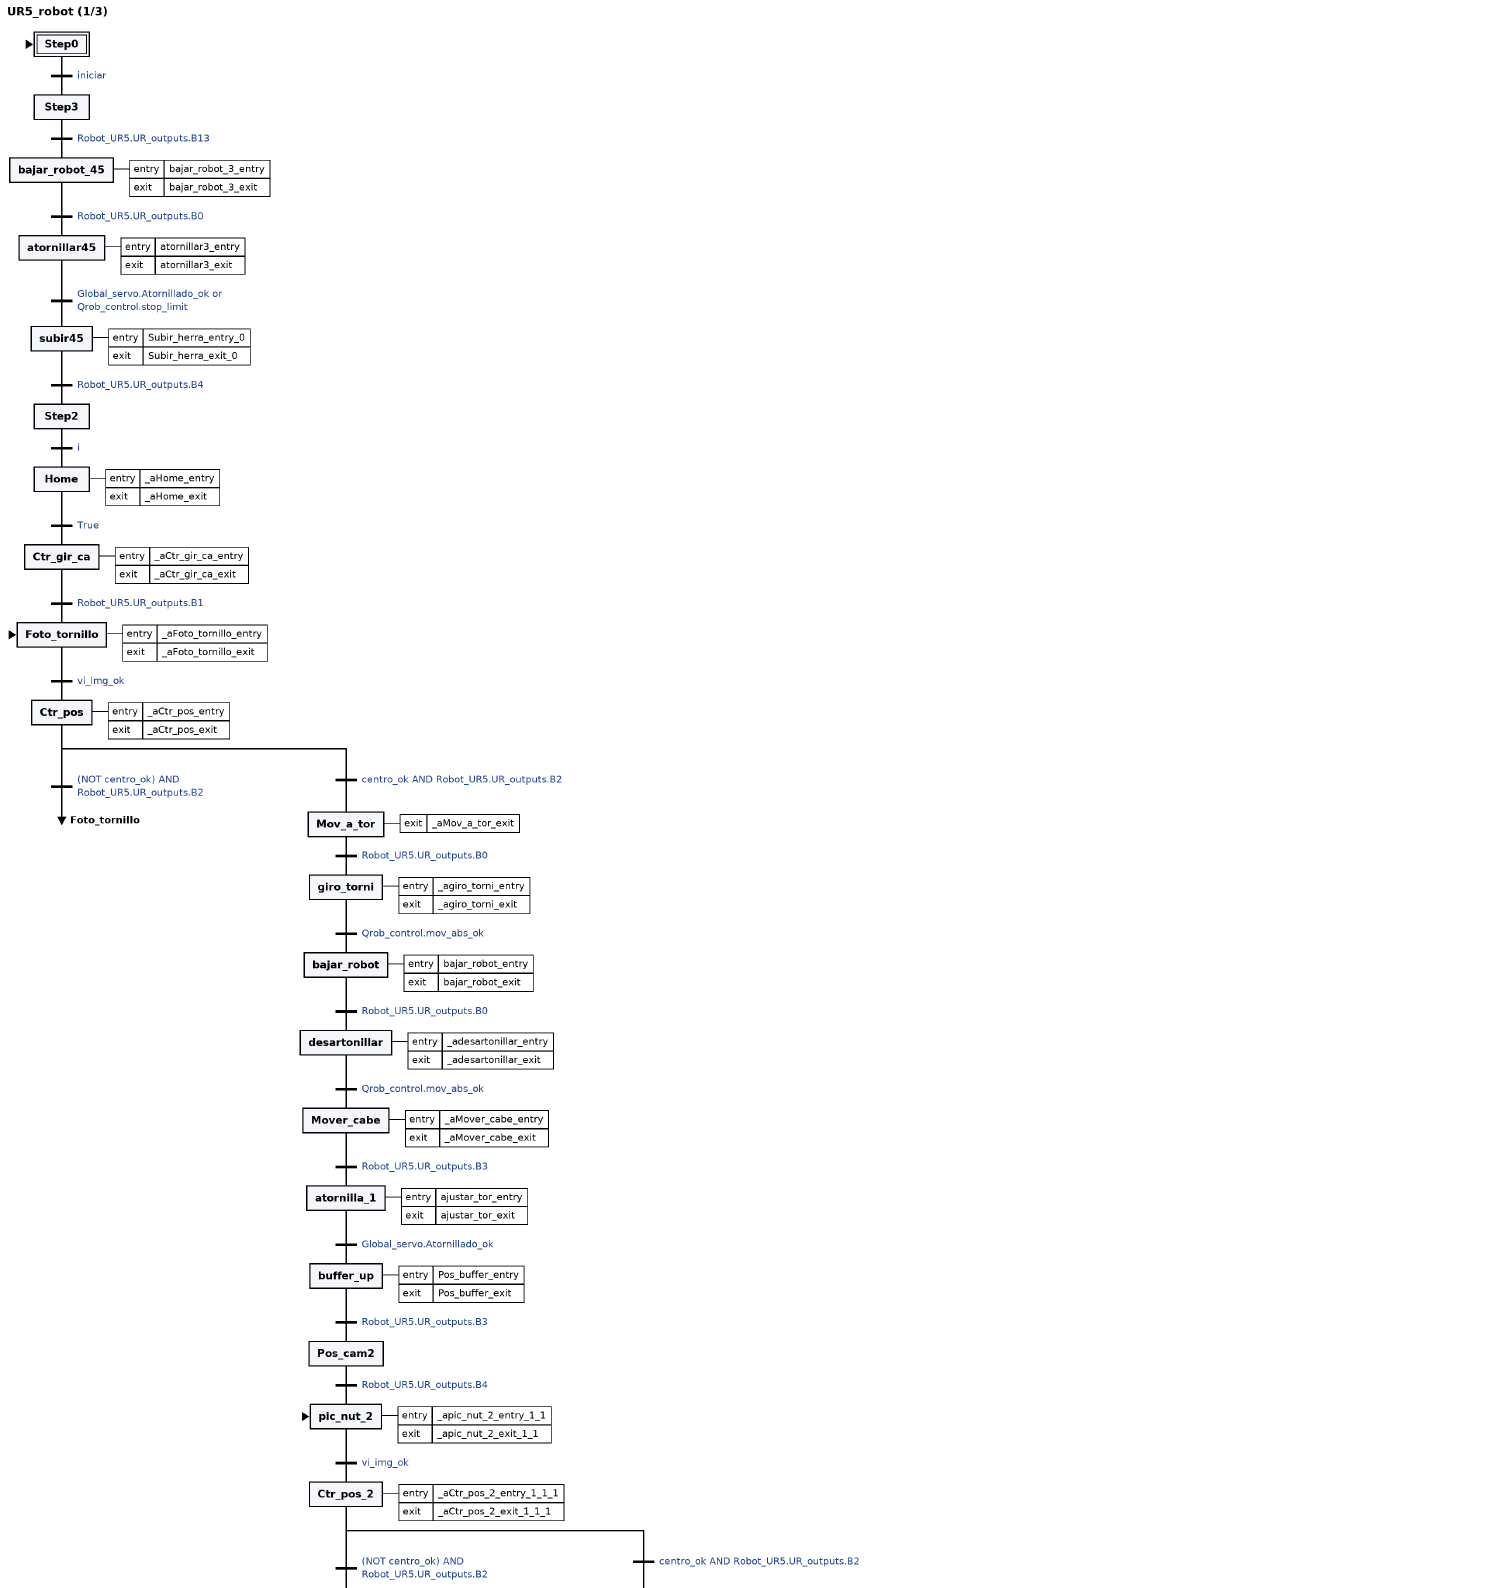
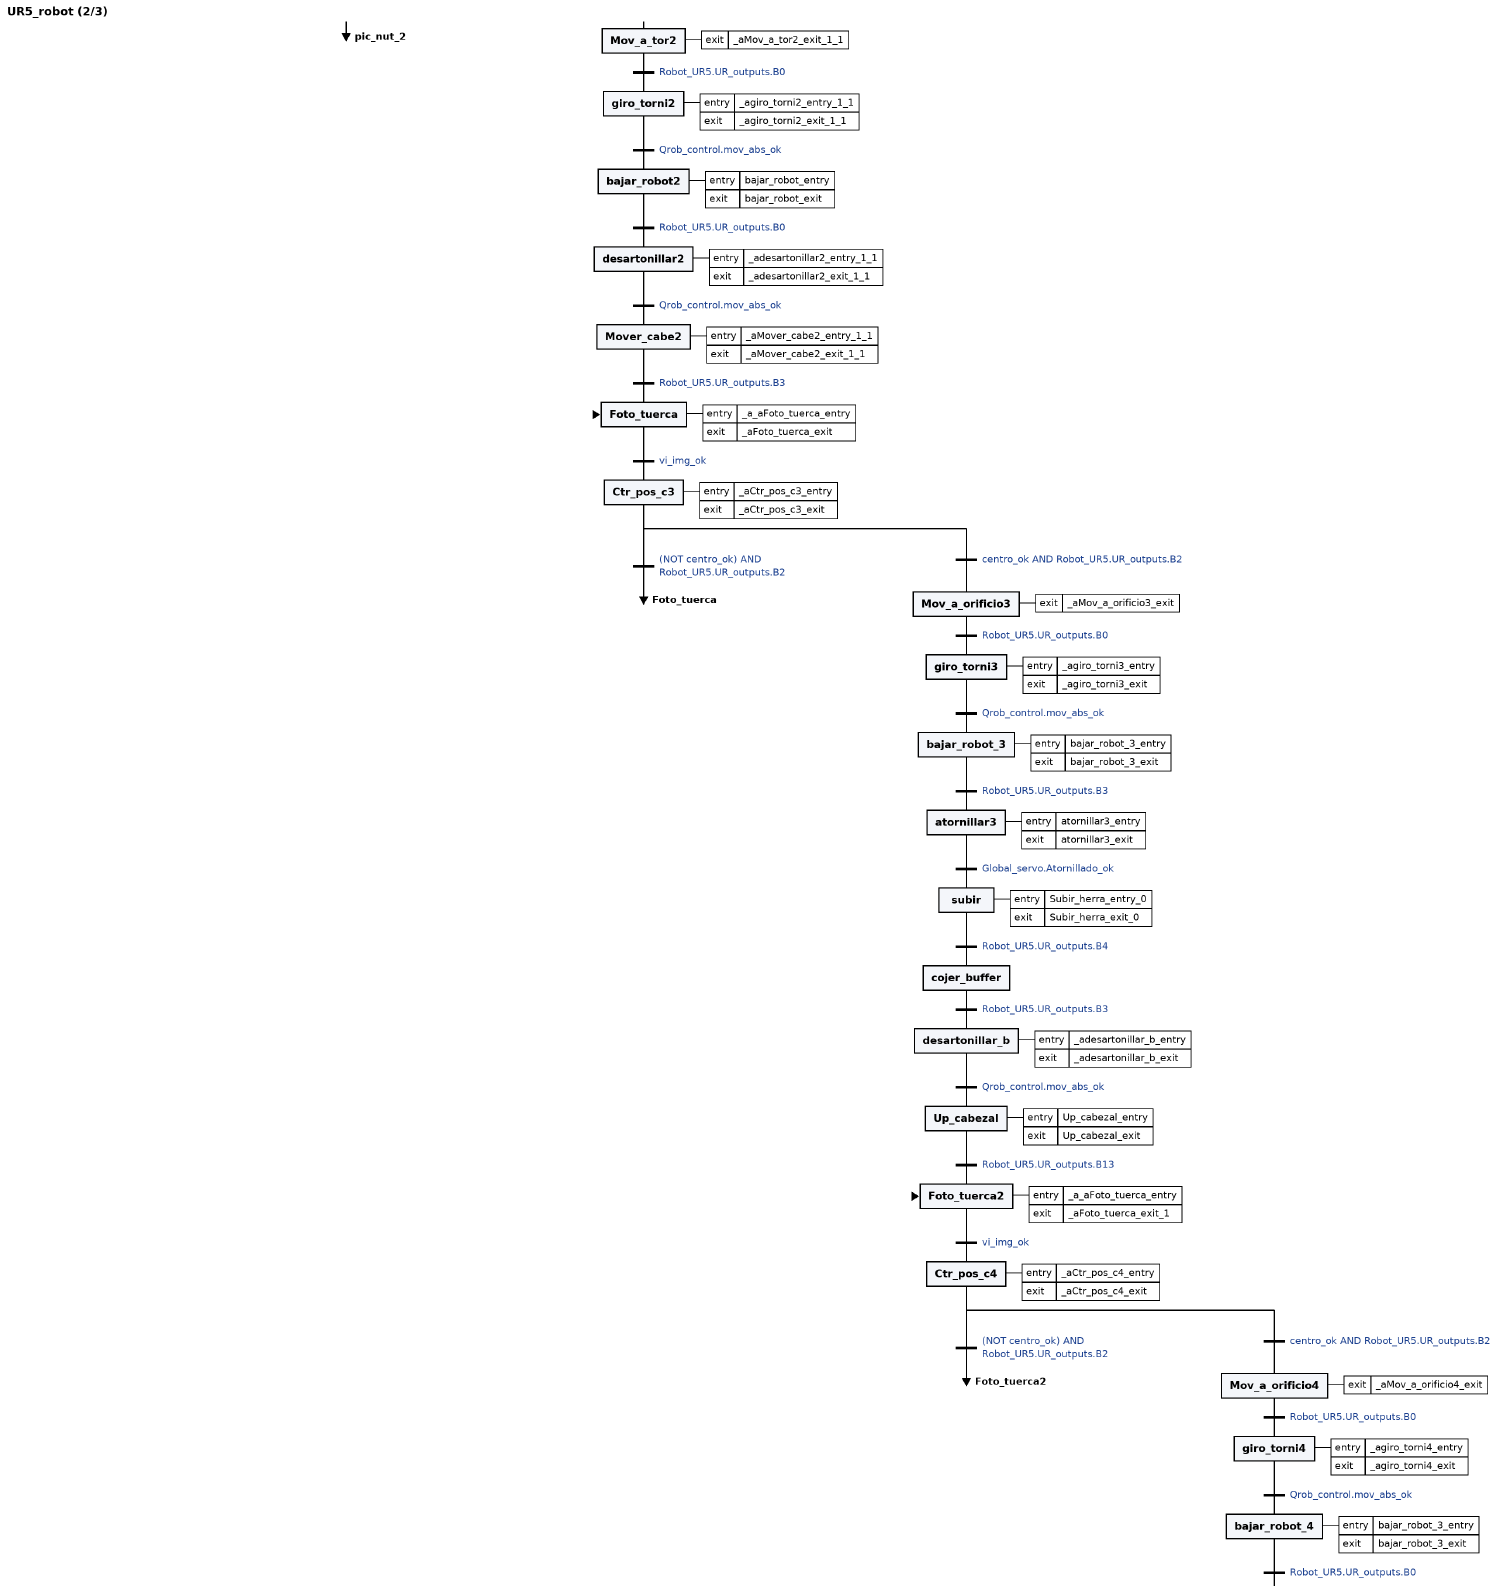
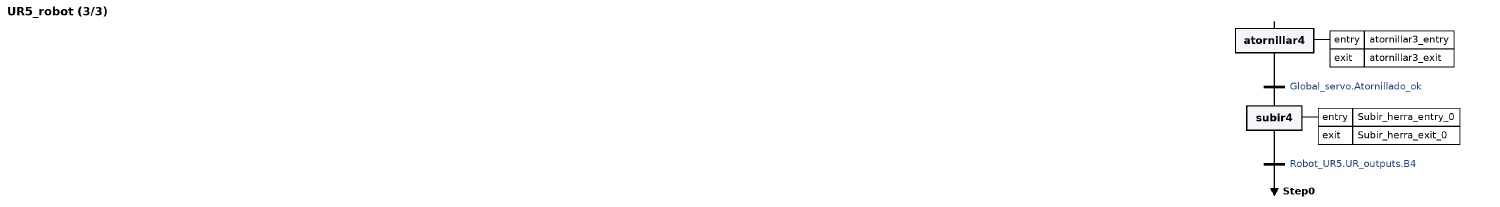
INITIAL_STEP Step0:
END_STEP
TRANSITION FROM Step0 TO Step3
    := iniciar;
END_TRANSITION
// macro Macro0 begins
STEP Step3:
END_STEP
TRANSITION FROM Step3 TO bajar_robot_45
    := Robot_UR5.UR_outputs.B13;
END_TRANSITION
STEP bajar_robot_45:
    bajar_robot_3_entry(P1);  // entry action
    bajar_robot_3_exit(P0);  // exit action
END_STEP
TRANSITION FROM bajar_robot_45 TO atornillar45
    := Robot_UR5.UR_outputs.B0;
END_TRANSITION
STEP atornillar45:
    atornillar3_entry(P1);  // entry action
    atornillar3_exit(P0);  // exit action
END_STEP
TRANSITION FROM atornillar45 TO subir45
    := Global_servo.Atornillado_ok or Qrob_control.stop_limit;
END_TRANSITION
STEP subir45:
    Subir_herra_entry_0(P1);  // entry action
    Subir_herra_exit_0(P0);  // exit action
END_STEP
TRANSITION FROM subir45 TO Step2
    := Robot_UR5.UR_outputs.B4;
END_TRANSITION
STEP Step2:
END_STEP
TRANSITION FROM Step2 TO Home
    := i;
END_TRANSITION
STEP Home:
    _aHome_entry(P1);  // entry action
    _aHome_exit(P0);  // exit action
END_STEP
TRANSITION FROM Home TO Ctr_gir_ca
    := True;
END_TRANSITION
STEP Ctr_gir_ca:
    _aCtr_gir_ca_entry(P1);  // entry action
    _aCtr_gir_ca_exit(P0);  // exit action
END_STEP
TRANSITION FROM Ctr_gir_ca TO Foto_tornillo
    := Robot_UR5.UR_outputs.B1;
END_TRANSITION
STEP Foto_tornillo:
    _aFoto_tornillo_entry(P1);  // entry action
    _aFoto_tornillo_exit(P0);  // exit action
END_STEP
TRANSITION FROM Foto_tornillo TO Ctr_pos
    := vi_img_ok;
END_TRANSITION
STEP Ctr_pos:
    _aCtr_pos_entry(P1);  // entry action
    _aCtr_pos_exit(P0);  // exit action
END_STEP
TRANSITION FROM Ctr_pos TO Foto_tornillo
    := (NOT centro_ok) AND Robot_UR5.UR_outputs.B2;
END_TRANSITION
TRANSITION FROM Ctr_pos TO Mov_a_tor
    := centro_ok AND Robot_UR5.UR_outputs.B2;
END_TRANSITION
STEP Mov_a_tor:
    _aMov_a_tor_exit(P0);  // exit action
END_STEP
TRANSITION FROM Mov_a_tor TO giro_torni
    := Robot_UR5.UR_outputs.B0;
END_TRANSITION
STEP giro_torni:
    _agiro_torni_entry(P1);  // entry action
    _agiro_torni_exit(P0);  // exit action
END_STEP
TRANSITION FROM giro_torni TO bajar_robot
    := Qrob_control.mov_abs_ok;
END_TRANSITION
STEP bajar_robot:
    bajar_robot_entry(P1);  // entry action
    bajar_robot_exit(P0);  // exit action
END_STEP
TRANSITION FROM bajar_robot TO desartonillar
    := Robot_UR5.UR_outputs.B0;
END_TRANSITION
STEP desartonillar:
    _adesartonillar_entry(P1);  // entry action
    _adesartonillar_exit(P0);  // exit action
END_STEP
TRANSITION FROM desartonillar TO Mover_cabe
    := Qrob_control.mov_abs_ok;
END_TRANSITION
STEP Mover_cabe:
    _aMover_cabe_entry(P1);  // entry action
    _aMover_cabe_exit(P0);  // exit action
END_STEP
TRANSITION FROM Mover_cabe TO atornilla_1
    := Robot_UR5.UR_outputs.B3;
END_TRANSITION
STEP atornilla_1:
    ajustar_tor_entry(P1);  // entry action
    ajustar_tor_exit(P0);  // exit action
END_STEP
TRANSITION FROM atornilla_1 TO buffer_up
    := Global_servo.Atornillado_ok;
END_TRANSITION
STEP buffer_up:
    Pos_buffer_entry(P1);  // entry action
    Pos_buffer_exit(P0);  // exit action
END_STEP
TRANSITION FROM buffer_up TO Pos_cam2
    := Robot_UR5.UR_outputs.B3;
END_TRANSITION
STEP Pos_cam2:
END_STEP
TRANSITION FROM Pos_cam2 TO pic_nut_2
    := Robot_UR5.UR_outputs.B4;
END_TRANSITION
STEP pic_nut_2:
    _apic_nut_2_entry_1_1(P1);  // entry action
    _apic_nut_2_exit_1_1(P0);  // exit action
END_STEP
TRANSITION FROM pic_nut_2 TO Ctr_pos_2
    := vi_img_ok;
END_TRANSITION
STEP Ctr_pos_2:
    _aCtr_pos_2_entry_1_1_1(P1);  // entry action
    _aCtr_pos_2_exit_1_1_1(P0);  // exit action
END_STEP
TRANSITION FROM Ctr_pos_2 TO pic_nut_2
    := (NOT centro_ok) AND Robot_UR5.UR_outputs.B2;
END_TRANSITION
TRANSITION FROM Ctr_pos_2 TO Mov_a_tor2
    := centro_ok AND Robot_UR5.UR_outputs.B2;
END_TRANSITION
STEP Mov_a_tor2:
    _aMov_a_tor2_exit_1_1(P0);  // exit action
END_STEP
TRANSITION FROM Mov_a_tor2 TO giro_torni2
    := Robot_UR5.UR_outputs.B0;
END_TRANSITION
STEP giro_torni2:
    _agiro_torni2_entry_1_1(P1);  // entry action
    _agiro_torni2_exit_1_1(P0);  // exit action
END_STEP
TRANSITION FROM giro_torni2 TO bajar_robot2
    := Qrob_control.mov_abs_ok;
END_TRANSITION
STEP bajar_robot2:
    bajar_robot_entry(P1);  // entry action
    bajar_robot_exit(P0);  // exit action
END_STEP
TRANSITION FROM bajar_robot2 TO desartonillar2
    := Robot_UR5.UR_outputs.B0;
END_TRANSITION
STEP desartonillar2:
    _adesartonillar2_entry_1_1(P1);  // entry action
    _adesartonillar2_exit_1_1(P0);  // exit action
END_STEP
TRANSITION FROM desartonillar2 TO Mover_cabe2
    := Qrob_control.mov_abs_ok;
END_TRANSITION
STEP Mover_cabe2:
    _aMover_cabe2_entry_1_1(P1);  // entry action
    _aMover_cabe2_exit_1_1(P0);  // exit action
END_STEP
TRANSITION FROM Mover_cabe2 TO Foto_tuerca
    := Robot_UR5.UR_outputs.B3;
END_TRANSITION
STEP Foto_tuerca:
    _a_aFoto_tuerca_entry(P1);  // entry action
    _aFoto_tuerca_exit(P0);  // exit action
END_STEP
TRANSITION FROM Foto_tuerca TO Ctr_pos_c3
    := vi_img_ok;
END_TRANSITION
STEP Ctr_pos_c3:
    _aCtr_pos_c3_entry(P1);  // entry action
    _aCtr_pos_c3_exit(P0);  // exit action
END_STEP
TRANSITION FROM Ctr_pos_c3 TO Foto_tuerca
    := (NOT centro_ok) AND Robot_UR5.UR_outputs.B2;
END_TRANSITION
TRANSITION FROM Ctr_pos_c3 TO Mov_a_orificio3
    := centro_ok AND Robot_UR5.UR_outputs.B2;
END_TRANSITION
STEP Mov_a_orificio3:
    _aMov_a_orificio3_exit(P0);  // exit action
END_STEP
TRANSITION FROM Mov_a_orificio3 TO giro_torni3
    := Robot_UR5.UR_outputs.B0;
END_TRANSITION
STEP giro_torni3:
    _agiro_torni3_entry(P1);  // entry action
    _agiro_torni3_exit(P0);  // exit action
END_STEP
TRANSITION FROM giro_torni3 TO bajar_robot_3
    := Qrob_control.mov_abs_ok;
END_TRANSITION
STEP bajar_robot_3:
    bajar_robot_3_entry(P1);  // entry action
    bajar_robot_3_exit(P0);  // exit action
END_STEP
TRANSITION FROM bajar_robot_3 TO atornillar3
    := Robot_UR5.UR_outputs.B3;
END_TRANSITION
STEP atornillar3:
    atornillar3_entry(P1);  // entry action
    atornillar3_exit(P0);  // exit action
END_STEP
TRANSITION FROM atornillar3 TO subir
    := Global_servo.Atornillado_ok;
END_TRANSITION
STEP subir:
    Subir_herra_entry_0(P1);  // entry action
    Subir_herra_exit_0(P0);  // exit action
END_STEP
TRANSITION FROM subir TO cojer_buffer
    := Robot_UR5.UR_outputs.B4;
END_TRANSITION
STEP cojer_buffer:
END_STEP
TRANSITION FROM cojer_buffer TO desartonillar_b
    := Robot_UR5.UR_outputs.B3;
END_TRANSITION
STEP desartonillar_b:
    _adesartonillar_b_entry(P1);  // entry action
    _adesartonillar_b_exit(P0);  // exit action
END_STEP
TRANSITION FROM desartonillar_b TO Up_cabezal
    := Qrob_control.mov_abs_ok;
END_TRANSITION
STEP Up_cabezal:
    Up_cabezal_entry(P1);  // entry action
    Up_cabezal_exit(P0);  // exit action
END_STEP
TRANSITION FROM Up_cabezal TO Foto_tuerca2
    := Robot_UR5.UR_outputs.B13;
END_TRANSITION
STEP Foto_tuerca2:
    _a_aFoto_tuerca_entry(P1);  // entry action
    _aFoto_tuerca_exit_1(P0);  // exit action
END_STEP
TRANSITION FROM Foto_tuerca2 TO Ctr_pos_c4
    := vi_img_ok;
END_TRANSITION
STEP Ctr_pos_c4:
    _aCtr_pos_c4_entry(P1);  // entry action
    _aCtr_pos_c4_exit(P0);  // exit action
END_STEP
TRANSITION FROM Ctr_pos_c4 TO Foto_tuerca2
    := (NOT centro_ok) AND Robot_UR5.UR_outputs.B2;
END_TRANSITION
TRANSITION FROM Ctr_pos_c4 TO Mov_a_orificio4
    := centro_ok AND Robot_UR5.UR_outputs.B2;
END_TRANSITION
STEP Mov_a_orificio4:
    _aMov_a_orificio4_exit(P0);  // exit action
END_STEP
TRANSITION FROM Mov_a_orificio4 TO giro_torni4
    := Robot_UR5.UR_outputs.B0;
END_TRANSITION
STEP giro_torni4:
    _agiro_torni4_entry(P1);  // entry action
    _agiro_torni4_exit(P0);  // exit action
END_STEP
TRANSITION FROM giro_torni4 TO bajar_robot_4
    := Qrob_control.mov_abs_ok;
END_TRANSITION
STEP bajar_robot_4:
    bajar_robot_3_entry(P1);  // entry action
    bajar_robot_3_exit(P0);  // exit action
END_STEP
TRANSITION FROM bajar_robot_4 TO atornillar4
    := Robot_UR5.UR_outputs.B0;
END_TRANSITION
STEP atornillar4:
    atornillar3_entry(P1);  // entry action
    atornillar3_exit(P0);  // exit action
END_STEP
TRANSITION FROM atornillar4 TO subir4
    := Global_servo.Atornillado_ok;
END_TRANSITION
STEP subir4:
    Subir_herra_entry_0(P1);  // entry action
    Subir_herra_exit_0(P0);  // exit action
END_STEP
TRANSITION FROM subir4 TO Step0
    := Robot_UR5.UR_outputs.B4;
END_TRANSITION

ACTION _a_aFoto_tuerca_entry:


vi_get_img_tuerca := True;
END_ACTION

ACTION _aCtr_gir_ca_entry:
Robot_UR5.UR_inputs.Floats.FLOAT3 := flip_real(data_to_robot.head_roll_right);
Robot_UR5.UR_inputs.Floats.FLOAT4 := flip_real(data_to_robot.head_roll_left);
Robot_UR5.UR_inputs.Bits.B0 := TRUE;
END_ACTION

ACTION _aCtr_gir_ca_exit:
Robot_UR5.UR_inputs.Bits.B0 := False;
END_ACTION

ACTION _aCtr_pos_2_entry_1_1_1:
vi_img_ok := FALSE;

Robot_UR5.UR_inputs.Floats.FLOAT0 := flip_real(cx);
Robot_UR5.UR_inputs.Floats.FLOAT1 := flip_real(cy);
Robot_UR5.UR_inputs.Floats.FLOAT2 := flip_real(giro);


IF ( ABS(cx) < 1) AND ( ABS(cy) < 1) THEN 
Robot_UR5.UR_inputs.Bits.B3 := TRUE;
centro_ok := TRUE;
ELSE 
Robot_UR5.UR_inputs.Bits.B3 := FALSE;
centro_ok := FALSE;	
END_IF

Robot_UR5.UR_inputs.Bits.B2 := TRUE;
END_ACTION

ACTION _aCtr_pos_2_exit_1_1_1:
Robot_UR5.UR_inputs.Bits.B2 := False;
END_ACTION

ACTION _aCtr_pos_c3_entry:
vi_img_ok := FALSE;

Robot_UR5.UR_inputs.Floats.FLOAT0 := flip_real(cx);
Robot_UR5.UR_inputs.Floats.FLOAT1 := flip_real(cy);



IF ( ABS(cx) < 0.5) AND ( ABS(cy) < 0.5) THEN 
Robot_UR5.UR_inputs.Bits.B3 := TRUE;
centro_ok := TRUE;
ELSE 
Robot_UR5.UR_inputs.Bits.B3 := FALSE;
centro_ok := FALSE;	
END_IF

Robot_UR5.UR_inputs.Bits.B2 := TRUE;
END_ACTION

ACTION _aCtr_pos_c3_exit:
Robot_UR5.UR_inputs.Bits.B2 := False;
END_ACTION

ACTION _aCtr_pos_c4_entry:
vi_img_ok := FALSE;

Robot_UR5.UR_inputs.Floats.FLOAT0 := flip_real(cx);
Robot_UR5.UR_inputs.Floats.FLOAT1 := flip_real(cy);



IF ( ABS(cx) < 0.5) AND ( ABS(cy) < 0.5) THEN 
Robot_UR5.UR_inputs.Bits.B3 := TRUE;
centro_ok := TRUE;
ELSE 
Robot_UR5.UR_inputs.Bits.B3 := FALSE;
centro_ok := FALSE;	
END_IF

Robot_UR5.UR_inputs.Bits.B2 := TRUE;
END_ACTION

ACTION _aCtr_pos_c4_exit:
Robot_UR5.UR_inputs.Bits.B2 := False;
END_ACTION

ACTION _aCtr_pos_entry:
vi_img_ok := FALSE;

Robot_UR5.UR_inputs.Floats.FLOAT0 := flip_real(cx);
Robot_UR5.UR_inputs.Floats.FLOAT1 := flip_real(cy);
Robot_UR5.UR_inputs.Floats.FLOAT2 := flip_real(giro);


IF ( ABS(cx) < 1) AND ( ABS(cy) < 1) THEN 
Robot_UR5.UR_inputs.Bits.B3 := TRUE;
centro_ok := TRUE;
ELSE 
Robot_UR5.UR_inputs.Bits.B3 := FALSE;
centro_ok := FALSE;	
END_IF

Robot_UR5.UR_inputs.Bits.B2 := TRUE;
END_ACTION

ACTION _aCtr_pos_exit:
Robot_UR5.UR_inputs.Bits.B2 := False;
END_ACTION

ACTION _adesartonillar_b_entry:




giro_desartonillado :=  (-24*360) + Qrob_control.actual_position;
Qrob_control.pos_mover_abs := giro_desartonillado;
Qrob_control.velocidad := 150;


Qrob_control.mover_abs := TRUE;
END_ACTION

ACTION _adesartonillar_b_exit:
Qrob_control.mover_abs := FALSE;
END_ACTION

ACTION _adesartonillar_entry:




giro_desartonillado := giro -(15*360);
//giro_desartonillado := giro -2160;
Qrob_control.pos_mover_abs := giro_desartonillado;
Qrob_control.velocidad := 150;


Qrob_control.mover_abs := TRUE;
END_ACTION

ACTION _adesartonillar_exit:
Qrob_control.mover_abs := FALSE;
END_ACTION

ACTION _adesartonillar2_entry_1_1:





giro_desartonillado := giro -(15*360);
//giro_desartonillado := giro -2160;
Qrob_control.pos_mover_abs := giro_desartonillado;
Qrob_control.velocidad := 150;


Qrob_control.mover_abs := TRUE;
END_ACTION

ACTION _adesartonillar2_exit_1_1:
Qrob_control.mover_abs := FALSE;
END_ACTION

ACTION _aFoto_tornillo_entry:
vi_get_img := True;
END_ACTION

ACTION _aFoto_tornillo_entry_1:
vi_get_img := True;
END_ACTION

ACTION _aFoto_tornillo_exit:
vi_get_img := False;
END_ACTION

ACTION _aFoto_tuerca_exit:

vi_get_img_tuerca := False;
END_ACTION

ACTION _aFoto_tuerca_exit_1:

vi_get_img_tuerca := False;
END_ACTION

ACTION _agiro_torni_entry:
//POU.detener := TRUE;
//Pou.detener := FALSE;


//home qrob while angle
giro_aux_int := ABS(TRUNC(Qrob_control.actual_position/360));
giro_aux_float := ABS( - (Qrob_control.actual_position/360));
giro_aux_float := -1*(giro_aux_float*360);






Qrob_control.velocidad := 50;
//Qrob_control.pos_mover_abs := giro;
Qrob_control.pos_mover_abs := (Qrob_control.actual_position + giro_aux_float) + giro;
Qrob_control.mover_abs := TRUE;
END_ACTION

ACTION _agiro_torni_exit:
Qrob_control.mover_abs := FALSE;
END_ACTION

ACTION _agiro_torni2_entry_1_1:
//POU.detener := TRUE;
//Pou.detener := FALSE;


//home qrob while angle
giro_aux_int := ABS(TRUNC(Qrob_control.actual_position/360));
giro_aux_float := ABS(giro_aux_int- (Qrob_control.actual_position/360));
giro_aux_float := -1*(giro_aux_float*360);






Qrob_control.velocidad := 50;
//Qrob_control.pos_mover_abs := giro;
Qrob_control.pos_mover_abs := (Qrob_control.actual_position + giro_aux_float) + giro;
giro := Qrob_control.pos_mover_abs;
Qrob_control.mover_abs := TRUE;
END_ACTION

ACTION _agiro_torni2_exit_1_1:
Qrob_control.mover_abs := FALSE;
END_ACTION

ACTION _agiro_torni3_entry:
//POU.detener := TRUE;
//Pou.detener := FALSE;


giro_aux_int := TRUNC(Qrob_control.actual_position/360);

giro_aux_float := ABS(giro_aux_int- (Qrob_control.actual_position/360));
giro_aux_float := -1*(giro_aux_float*360);

Qrob_control.velocidad := 100;
Qrob_control.pos_mover_abs := Qrob_control.actual_position + giro_aux_float;
Qrob_control.mover_abs := TRUE;
END_ACTION

ACTION _agiro_torni3_exit:
Qrob_control.mover_abs := FALSE;
END_ACTION

ACTION _agiro_torni4_entry:
//POU.detener := TRUE;
//Pou.detener := FALSE;

//Qrob_control.velocidad := 100;
//Qrob_control.pos_mover_abs := 0;
//Qrob_control.mover_abs := TRUE;


giro_aux_int := TRUNC(Qrob_control.actual_position/360);

giro_aux_float := ABS(giro_aux_int- (Qrob_control.actual_position/360));
giro_aux_float := -1*(giro_aux_float*360);

Qrob_control.velocidad := 100;
Qrob_control.pos_mover_abs := Qrob_control.actual_position + giro_aux_float;
Qrob_control.mover_abs := TRUE;
END_ACTION

ACTION _agiro_torni4_exit:
Qrob_control.mover_abs := FALSE;
END_ACTION

ACTION _aHome_entry:
i := FALSE;
Robot_UR5.UR_inputs.Bits.B0 := TRUE;
//POU.EnableAxis1 := True;
giro :=0;
//Qrob_control.ajustar_tornillo := FALSE;
//Qrob_control.pos_mover_abs := 0;
//Qrob_control.velocidad := 100;


//Qrob_control.mover_abs := TRUE;
END_ACTION

ACTION _aHome_exit:
Robot_UR5.UR_inputs.Bits.B0 := FALSE;
iniciar := FALSE;
Qrob_control.mover_abs := False;
END_ACTION

ACTION _aMov_a_orificio3_exit:
Robot_UR5.UR_inputs.Bits.B2 := FALSE;
END_ACTION

ACTION _aMov_a_orificio4_exit:
Robot_UR5.UR_inputs.Bits.B2 := FALSE;
END_ACTION

ACTION _aMov_a_tor_exit:
Robot_UR5.UR_inputs.Bits.B2 := FALSE;
END_ACTION

ACTION _aMov_a_tor2_exit_1_1:
Robot_UR5.UR_inputs.Bits.B2 := FALSE;
END_ACTION

ACTION _aMover_cabe_entry:
Robot_UR5.UR_inputs.Bits.B5 := True;
END_ACTION

ACTION _aMover_cabe_exit:
Robot_UR5.UR_inputs.Bits.B5 := False;
END_ACTION

ACTION _aMover_cabe2_entry_1_1:
Robot_UR5.UR_inputs.Bits.B5 := True;
END_ACTION

ACTION _aMover_cabe2_exit_1_1:
Robot_UR5.UR_inputs.Bits.B5 := False;
END_ACTION

ACTION _apic_nut_2_entry_1_1:
vi_get_img := True;
END_ACTION

ACTION _apic_nut_2_exit_1_1:
vi_get_img := False;
END_ACTION

ACTION ajustar_tor_entry:


//Atornillado_funcion(Iniciar:= TRUE, Corriente := 60, vueltas := 8, giro_alivio := 3);

Atornillar_CS.UR5.Corriente := 10;
Atornillar_CS.UR5.Vueltas := 21;
Atornillar_CS.UR5.Iniciar := TRUE;
END_ACTION

ACTION ajustar_tor_exit:
Global_servo.Atornillado_ok := FALSE;
Atornillar_CS.UR5.Iniciar := FALSE;
END_ACTION

ACTION atornillar_2_entry:

Atornillar_CS.UR5.Corriente :=100;
Atornillar_CS.UR5.Vueltas := 4;
Atornillar_CS.UR5.Iniciar := True;
END_ACTION

ACTION atornillar_2_exit:
Global_servo.Atornillado_ok := FALSE;
Atornillar_CS.UR5.Iniciar := False;
END_ACTION

ACTION atornillar3_entry:

//Atornillado_funcion(Iniciar:= TRUE, Corriente := 60, vueltas := 8, giro_alivio := 3);

//Atornillar_CS.UR5.Corriente := 75;
//Atornillar_CS.UR5.Vueltas := 13;
//Atornillar_CS.UR5.Iniciar := TRUE;

Qrob_control.ajustar_tornillo := TRUE;
Qrob_control.limite_corriente := 150;
Qrob_control.mover_horario := TRUE;
END_ACTION

ACTION atornillar3_exit:
//Global_servo.Atornillado_ok := FALSE;
//Atornillar_CS.UR5.Iniciar := FALSE;



Qrob_control.ajustar_tornillo := FALSE;
Qrob_control.limite_corriente := 100;
Qrob_control.mover_horario := FALSE;
Qrob_control.detener := FALSE;
END_ACTION

ACTION bajar_robot_3_entry:

Robot_UR5.UR_inputs.Bits.B0 := TRUE;
END_ACTION

ACTION bajar_robot_3_exit:
Robot_UR5.UR_inputs.Bits.B0 := FALSE;
Robot_UR5.UR_inputs.Bits.B10 := False;
END_ACTION

ACTION bajar_robot_entry:
Robot_UR5.UR_inputs.Bits.B0 := TRUE;
END_ACTION

ACTION bajar_robot_exit:
Robot_UR5.UR_inputs.Bits.B0 := False;
END_ACTION

ACTION Cabe_separador_entry:
Robot_UR5.UR_inputs.Bits.B5 := TRUE;
END_ACTION

ACTION Cabe_separador_exit:
Robot_UR5.UR_inputs.Bits.B5 := False;
END_ACTION

ACTION Pos_buffer_entry:

Robot_UR5.UR_inputs.Bits.B7 := TRUE;
END_ACTION

ACTION Pos_buffer_exit:

Robot_UR5.UR_inputs.Bits.B7 := False;
END_ACTION

ACTION Step1_entry:
Robot_UR5.UR_inputs.Bits.B7 := TRUE;
END_ACTION

ACTION Step1_exit:
Robot_UR5.UR_inputs.Bits.B7 := False;
END_ACTION

ACTION Subir_herra_entry:
Robot_UR5.UR_inputs.Bits.B7 := TRUE;
Qrob_control.detener := TRUE;
Qrob_control.detener := FALSE;


Robot_UR5.UR_inputs.Bits.B7 := TRUE;
Qrob_control.pos_mover_abs := Qrob_control.actual_position -10;




Qrob_control.velocidad := 1;
Qrob_control.mover_abs := TRUE;
END_ACTION

ACTION Subir_herra_entry_0:
Robot_UR5.UR_inputs.Bits.B5 := TRUE;
Robot_UR3.UR_outputs.B6 := False;
END_ACTION

ACTION Subir_herra_exit:
Robot_UR5.UR_inputs.Bits.B7 := FALSE;
Qrob_control.mover_abs := FALSE;
END_ACTION

ACTION Subir_herra_exit_0:
Robot_UR5.UR_inputs.Bits.B5 := FALSE;
Robot_UR3.UR_outputs.B6 := True;
END_ACTION

ACTION Up_cabezal_entry:
Robot_UR5.UR_inputs.Bits.B8 := TRUE;
END_ACTION

ACTION Up_cabezal_exit:
Robot_UR5.UR_inputs.Bits.B8 := False;
END_ACTION

END_PROGRAM
